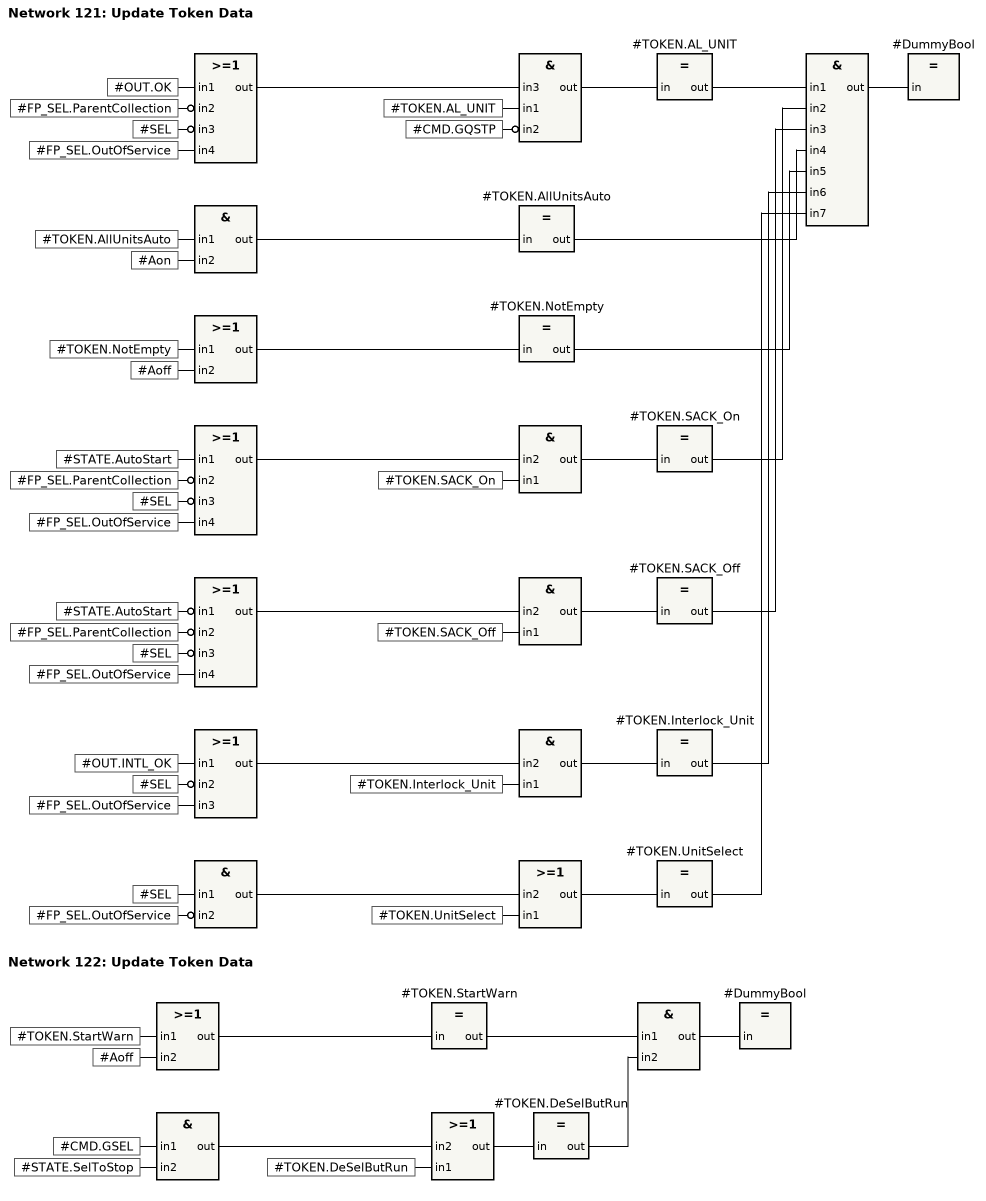
   #TOKEN.AL_UNIT := (#OUT.OK OR NOT #FP_SEL.ParentCollection OR NOT #SEL OR #FP_SEL.OutOfService) AND #TOKEN.AL_UNIT AND NOT #CMD.GQSTP;
   #TOKEN.SACK_On := (#STATE.AutoStart OR NOT #FP_SEL.ParentCollection OR NOT #SEL OR #FP_SEL.OutOfService) AND #TOKEN.SACK_On;
   #TOKEN.SACK_Off := (NOT #STATE.AutoStart OR NOT #FP_SEL.ParentCollection OR NOT #SEL OR #FP_SEL.OutOfService) AND #TOKEN.SACK_Off;
   #TOKEN.AllUnitsAuto := #TOKEN.AllUnitsAuto AND #Aon;
   #TOKEN.NotEmpty := #TOKEN.NotEmpty OR #Aoff;
   #TOKEN.Interlock_Unit := (#OUT.INTL_OK OR NOT #SEL OR #FP_SEL.OutOfService) AND #TOKEN.Interlock_Unit;
   #TOKEN.UnitSelect := (#SEL AND NOT #FP_SEL.OutOfService) OR #TOKEN.UnitSelect;
   #DummyBool := #TOKEN.AL_UNIT AND #TOKEN.SACK_On AND #TOKEN.SACK_Off AND #TOKEN.AllUnitsAuto AND #TOKEN.NotEmpty AND #TOKEN.Interlock_Unit AND #TOKEN.UnitSelect;
END_REGION

REGION Network 122: Update Token Data
   #TOKEN.StartWarn := #TOKEN.StartWarn OR #Aoff;
   #TOKEN.DeSelButRun := (#CMD.GSEL AND #STATE.SelToStop) OR #TOKEN.DeSelButRun;
   #DummyBool := #TOKEN.StartWarn AND #TOKEN.DeSelButRun;
END_REGION

REGION Network 123: Interlock Status to HMI
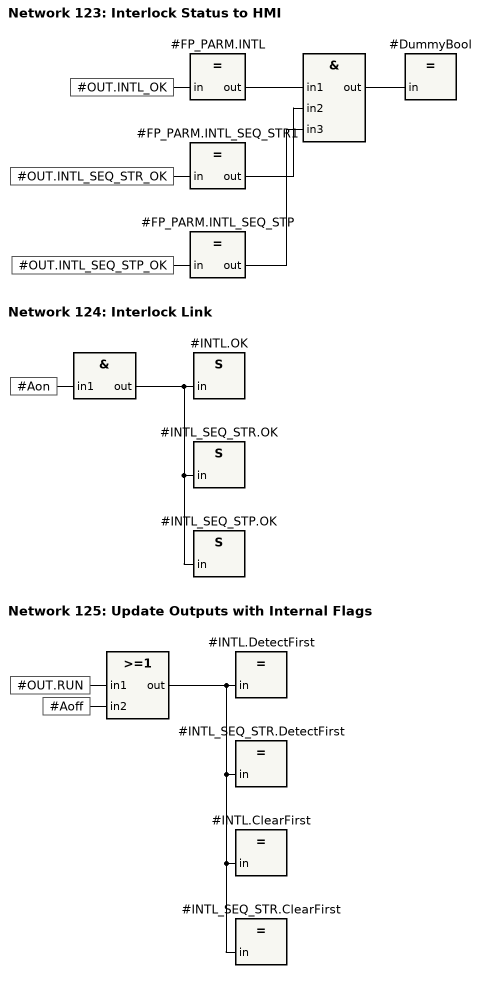
   #FP_PARM.INTL := #OUT.INTL_OK;
   #FP_PARM.INTL_SEQ_STR1 := #OUT.INTL_SEQ_STR_OK;
   #FP_PARM.INTL_SEQ_STP := #OUT.INTL_SEQ_STP_OK;
   #DummyBool := #OUT.INTL_OK AND #OUT.INTL_SEQ_STR_OK AND #OUT.INTL_SEQ_STP_OK;
END_REGION

REGION Network 124: Interlock Link
   IF #Aon THEN
       #INTL.OK := TRUE;
       #INTL_SEQ_STR.OK := TRUE;
       #INTL_SEQ_STP.OK := TRUE;
   END_IF;
END_REGION

REGION Network 125: Update Outputs with Internal Flags
   #INTL.DetectFirst := #OUT.RUN OR #Aoff;
   #INTL_SEQ_STR.DetectFirst := #INTL.DetectFirst;
   #INTL.ClearFirst := #INTL.DetectFirst;
   #INTL_SEQ_STR.ClearFirst := #INTL.DetectFirst;
END_REGION
END_FUNCTION_BLOCK

FUNCTION_BLOCK "ACESYS_BQ16_PROG"   // FB240, FBD
TITLE = ACESYS V8.0 - Build 002 - Air Blaster Program Block
{ S7_Optimized_Access := 'FALSE' }
AUTHOR : FLSmidth
FAMILY : ACESYS
NAME : Air_Prog
VERSION : 8.0
// This block is a separate program block for a airblaster and shall work as a 
// "child" for Air-blaster control block, ACESYS_BQ16_CTRL
// Data to the control block shall be send in a data structure: BQ16_Link (UDT224)
   VAR_OUTPUT
      Run : Bool;   // Program Running
      MSW : "ACESYS_HMI_STAT_32T";
   END_VAR
   VAR_IN_OUT
      TOKEN : "ACESYS_TOKEN";
      ProgLink : "ACESYS_BQ16";   // Link Command unit <-> Program Unit
   END_VAR
   VAR
      BlockInfo : Struct
         ACESYS_Version : Int;   // Block Version
         ACESYS_Build : Int;   // Block Build Number
         DB_Number : Int;
      END_STRUCT;
      FP_CMD : Struct   // Faceplate Commands
         Previous : Bool;   // FacePlateCmd (bit 8): Previous Sequence
         Next : Bool;   // FacePlateCmd (bit 9): Next Sequence
         Spare_Bool_01 : Bool;   // FacePlateCmd (bit 10): Spare
         Spare_Bool_02 : Bool;   // FacePlateCmd (bit 11): Spare
         Spare_Bool_03 : Bool;   // FacePlateCmd (bit 12): Spare
         Spare_Bool_04 : Bool;   // FacePlateCmd (bit 13): Spare
         Spare_Bool_05 : Bool;   // FacePlateCmd (bit 14): Spare
         Spare_Bool_06 : Bool;   // FacePlateCmd (bit 15): ECS Acknowledge
         Spare_Bool_07 : Bool;   // FacePlateCmd (bit 0): Spare
         Spare_Bool_08 : Bool;   // FacePlateCmd (bit 1): Spare
         Spare_Bool_09 : Bool;   // FacePlateCmd (bit 2): Spare
         Spare_Bool_10 : Bool;   // FacePlateCmd (bit 3): Spare
         Spare_Bool_11 : Bool;   // FacePlateCmd (bit 4): Spare
         Spare_Bool_12 : Bool;   // FacePlateCmd (bit 5): Spare
         Spare_Bool_13 : Bool;   // FacePlateCmd (bit 6): Spare
         Spare_Bool_14 : Bool;   // FacePlateCmd (bit 7): Spare
      END_STRUCT;
      FP_DIM : Struct   // Faceplate Dimmed Buttons
         Previous : Bool;   // Dimout Prev button to ECS
         Next : Bool;   // Dimout Next button to ECS
         Spare_Bool_01 : Bool;
         Spare_Bool_02 : Bool;
         Spare_Bool_03 : Bool;
         Spare_Bool_04 : Bool;
         Spare_Bool_05 : Bool;
         Spare_Bool_06 : Bool;
         Spare_Bool_07 : Bool;
         Spare_Bool_08 : Bool;
         Spare_Bool_09 : Bool;
         Spare_Bool_10 : Bool;
         Spare_Bool_11 : Bool;
         Spare_Bool_12 : Bool;
         Spare_Bool_13 : Bool;
         Spare_Bool_14 : Bool;
      END_STRUCT;
      FP_PARM : Struct
         ProgNo : Int;   // Program Number to Faceplate
         SEQNO : Int;   // Sequence No in Matrix Configuration Faceplate
         NumberBlasters : Int := 16;   // Number Of Blasters to be Used
         NumberSteps : Int := 16;   // Number Of Steps to be Used
         Blast_Stp_Dyn01 : Bool;   // Blaster 1 Setup Dynamic bit to ECS
         Blast_Stp_Dyn02 : Bool;   // Blaster 2 Setup Dynamic bit to ECS
         Blast_Stp_Dyn03 : Bool;   // Blaster 3 Setup Dynamic bit to ECS
         Blast_Stp_Dyn04 : Bool;   // Blaster 4 Setup Dynamic bit to ECS
         Blast_Stp_Dyn05 : Bool;   // Blaster 5 Setup Dynamic bit to ECS
         Blast_Stp_Dyn06 : Bool;   // Blaster 6 Setup Dynamic bit to ECS
         Blast_Stp_Dyn07 : Bool;   // Blaster 7 Setup Dynamic bit to ECS
         Blast_Stp_Dyn08 : Bool;   // Blaster 8 Setup Dynamic bit to ECS
         Blast_Stp_Dyn09 : Bool;   // Blaster 9 Setup Dynamic bit to ECS
         Blast_Stp_Dyn10 : Bool;   // Blaster 10 Setup Dynamic bit to ECS
         Blast_Stp_Dyn11 : Bool;   // Blaster 11 Setup Dynamic bit to ECS
         Blast_Stp_Dyn12 : Bool;   // Blaster 12 Setup Dynamic bit to ECS
         Blast_Stp_Dyn13 : Bool;   // Blaster 13 Setup Dynamic bit to ECS
         Blast_Stp_Dyn14 : Bool;   // Blaster 14 Setup Dynamic bit to ECS
         Blast_Stp_Dyn15 : Bool;   // Blaster 15 Setup Dynamic bit to ECS
         Blast_Stp_Dyn16 : Bool;   // Blaster 16 Setup Dynamic bit to ECS
         CurrentState : Array[1..16] of Int;   // Blaster State for ECS animation
      END_STRUCT;
      FP_PARM_CycleTime : Array[1..6] of Int;   // SP from FP
      FP_PARM_OffsetTime : Array[1..6] of Int;   // SP from FP
      FP_PARM_PulseTime : Array[1..6] of Int;   // SP from FP
      FP_PARM_StepTime : Array[1..6] of Int;   // SP from FP
      FP_PARM_Blaster_SEQNO : Array[1..16] of Int;   // Blaster Configured Sequence
      FP_PARM_BlastSEQX_Setup : Array[1..16] of Word;   // Blaster Setup From/To ECS
      FP_PARM_Blaster_Step : Array[1..16] of Word;   // Blaster Configurated Step Mask
      FP_PARM_MaxNumberSteps : Array[1..16] of Int;   // Max Step to be executed with current Time constants
      FP_PARM_PauseTime : Array[1..16] of Int;   // Time until next Cycle
      FP_PARM_MaxStep : Array[1..6] of Int;   // Max Step to be executed with current Time constants
      FP_PARM_OffsetStep : Array[1..16] of Bool;
      BlastSEQ1_Setup : Array[1..16] of Word;   // Blaster Setup in sequence 01
      BlastSEQ2_Setup : Array[1..16] of Word;   // Blaster Setup in sequence 02
      BlastSEQ3_Setup : Array[1..16] of Word;   // Blaster Setup in sequence 03
      BlastSEQ4_Setup : Array[1..16] of Word;   // Blaster Setup in sequence 04
      BlastSEQ5_Setup : Array[1..16] of Word;   // Blaster Setup in sequence 05
      BlastSEQ6_Setup : Array[1..16] of Word;   // Blaster Setup in sequence 06
      BlastSEQ_CycleTime_Mem : Array[1..6] of Int;   // Internal Timer Value
      BlastSEQ_CycleTime_PV : Array[1..6] of Int;   // For Next Blast, Time Calculation
      StepTime_PV : Array[1..6] of Int;   // For Next Blast, Time Calculation
      SEQTmr_SP : Array[1..6] of Int;   // For Next Blast, Time Calculation
      BlastSEQ_State : Array[1..6] of Word;   // Actual Step Mask of the Sequence
      TimeACT_PV : Array[1..6] of Int;   // For Next Blast, Time Calculation
      PauseTime : Array[1..6] of Int;   // Time until next Cycle
      BlastSEQ_CycleTime_DN : Array[1..6] of Bool;   // Timer Done
      StepSEQ_Offset : Array[1..6] of Bool;   // Select Offset time
      StepSEQ_Pulse : Array[1..6] of Bool;   // Select Pulse Time
      StepSEQ_Step : Array[1..6] of Bool;   // Select Step Time
      StepSEQ_Done : Array[1..6] of Bool;   // Step Sequence Done
      BlastSEQ_Start : Array[1..6] of Bool;   // Start Sequence
      BlastSEQ_EN : Array[1..6] of Bool;   // Pause the Execution of sequence
      InOffset_Pause : Array[1..6] of Bool;   // Pause the Execution of sequence
      CycleInStep : Array[1..6] of Bool;   // Cycle is running a step
      SequenceInOffset : Array[1..6] of Bool;   // Sequence is in Offset state
      TimeOLD : Array[1..6] of Time;
      TimeACT : Array[1..6] of Time;
      TimeSP : Array[1..6] of Time;
      SEQ_Old_Config : Array[1..6] of DWord;
      CycleTime_Old : Array[1..6] of Int;
      OffsetTime_Old : Array[1..6] of Int;
      PulseTime_Old : Array[1..6] of Int;
      StepTime_Old : Array[1..6] of Int;
      ConfigChanged : Bool;   // Configuration Changed Status
      ProgLink_Start : Bool;   // Start from Control Block
      ProgLink_Reset : Bool;   // Reset Sequence Option from Control Block
      Run_Delay : Bool;   // One scan delayed RUN signal
      SEQ01_Timer_DN : Bool;
      SEQ02_Timer_DN : Bool;
      SEQ03_Timer_DN : Bool;
      SEQ04_Timer_DN : Bool;
      SEQ05_Timer_DN : Bool;
      SEQ06_Timer_DN : Bool;
      Old_SEQNO : Int;
      StatusWork : Int;
      MSW_Status : Int;
      SYNC_TIME : Struct
         Mem : Int;
         PRE : Int;
         PRE_Old : Int;
         PV : Int;
         DN : Bool;
         TT : Bool;
      END_STRUCT;
      CMD_Int : Struct
         Previous : Bool;
         Next : Bool;
      END_STRUCT;
      ONS : Struct
         Previous : Bool;
         Next : Bool;
         Pulse : Array[1..6] of Bool;   // Pause the Execution of sequence
         Pulse1 : Array[1..6] of Bool;   // Pause the Execution of sequence
         ConfigChanged : Bool;
         BlastSEQ01_Start : Bool;
         BlastSEQ02_Start : Bool;
         BlastSEQ03_Start : Bool;
         BlastSEQ04_Start : Bool;
         BlastSEQ05_Start : Bool;
         BlastSEQ06_Start : Bool;
         Sync_Time_DN : Bool;
      END_STRUCT;
      OUT : Struct
         Run : Bool;
      END_STRUCT;
      SEQ01_Timer : TON_TIME;
      SEQ02_Timer : TON_TIME;
      SEQ03_Timer : TON_TIME;
      SEQ04_Timer : TON_TIME;
      SEQ05_Timer : TON_TIME;
      SEQ06_Timer : TON_TIME;
   END_VAR
   VAR_TEMP
      Aon : Bool;
      Aoff : Bool;
      DummyBool : Bool;
      DummyBool1 : Bool;
      DummyTime : Time;
      DummyWord : Word;
      DummyDint : DInt;
      DummyInt : Int;
      DummyReal : Real;
      DummyReal1 : Real;
      Current_SEQNO : Int;
      NextTime_BlastLoop : Int;
      Offset_Int : Int;
      NXT_SEQ_State : Word;   // Current Step Mask of the Sequence
      NXT_SEQ_PULSE : Bool;
      SEQ_Current_Config : Array[1..6] of DWord;
      ClearBlasterLoop : Int;
      ClearStepLoop : Int;
      StepMask : Word;   // Allowed Steps set to 1
      ChangeConfigLoop : Int;
   END_VAR
   VAR_TEMP   // added for the SCL form of the ladder/FBD networks
      _w1 : Bool;
      _w2 : Bool;
      _w3 : Bool;
      _w4 : Bool;
      _w5 : Bool;
      _w6 : Bool;
      _w7 : Bool;
      _w8 : Bool;
      _w9 : Bool;
      _w10 : Bool;
      _w11 : Bool;
      _w12 : Bool;
      _w13 : Bool;
      _w14 : Bool;
      _w15 : Bool;
      _w16 : Bool;
   END_VAR
   // FP_PARM_CycleTime[1] := 1;
   // FP_PARM_CycleTime[2] := 1;
   // FP_PARM_CycleTime[3] := 1;
   // FP_PARM_CycleTime[4] := 1;
   // FP_PARM_CycleTime[5] := 1;
   // FP_PARM_CycleTime[6] := 1;
   // FP_PARM_OffsetTime[1] := 30;
   // FP_PARM_OffsetTime[2] := 30;
   // FP_PARM_OffsetTime[3] := 30;
   // FP_PARM_OffsetTime[4] := 30;
   // FP_PARM_OffsetTime[5] := 30;
   // FP_PARM_OffsetTime[6] := 30;
   // FP_PARM_PulseTime[1] := 500;
   // FP_PARM_PulseTime[2] := 500;
   // FP_PARM_PulseTime[3] := 500;
   // FP_PARM_PulseTime[4] := 500;
   // FP_PARM_PulseTime[5] := 500;
   // FP_PARM_PulseTime[6] := 500;
   // FP_PARM_StepTime[1] := 5;
   // FP_PARM_StepTime[2] := 5;
   // FP_PARM_StepTime[3] := 5;
   // FP_PARM_StepTime[4] := 5;
   // FP_PARM_StepTime[5] := 5;
   // FP_PARM_StepTime[6] := 5;
BEGIN

REGION Network 1: Aon/Aoff Definition
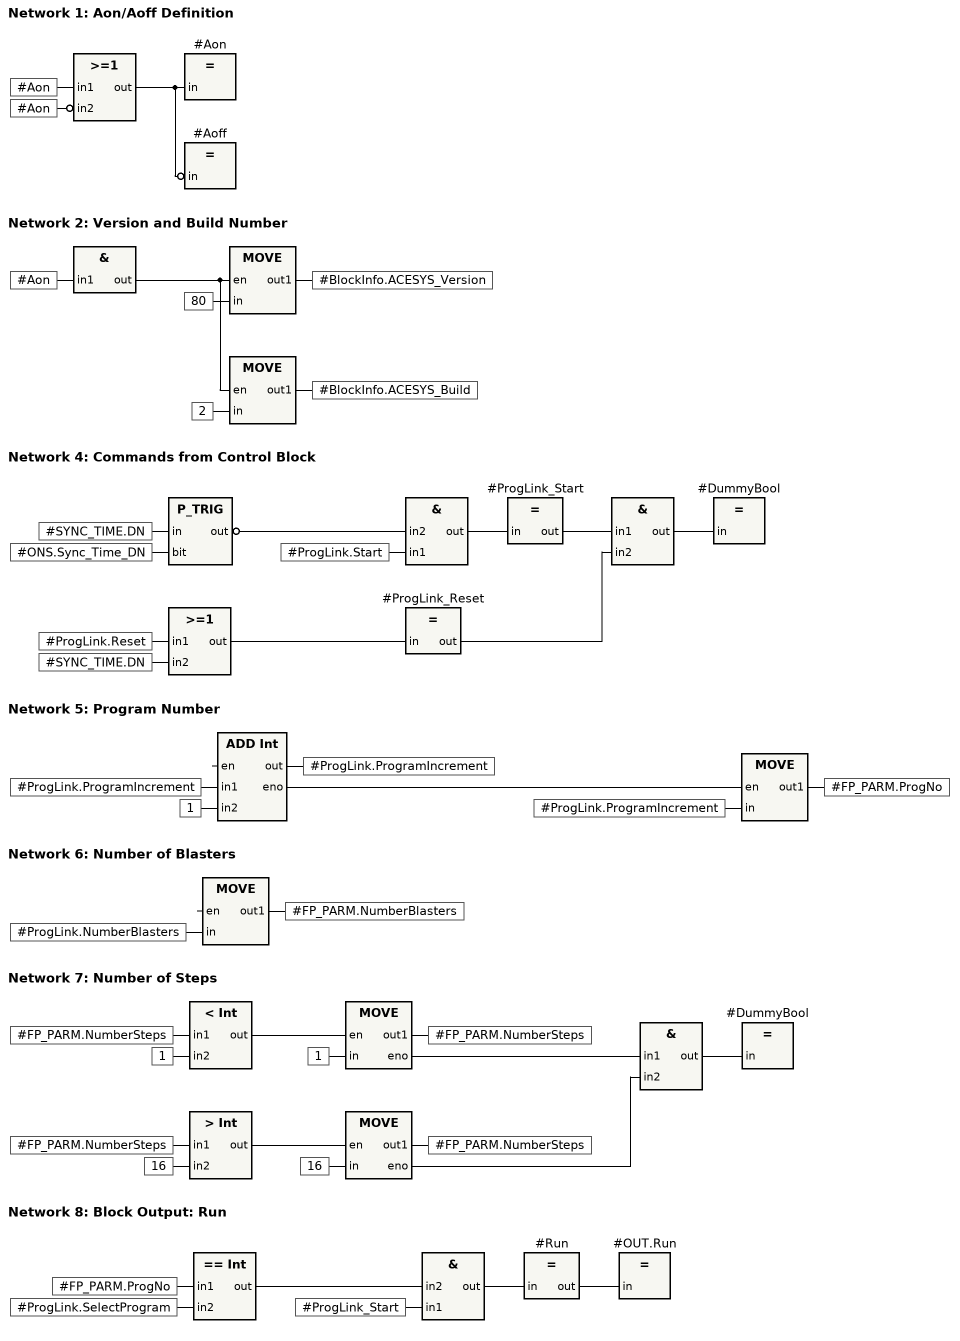
   #Aon := #Aon OR NOT #Aon;
   #Aoff := NOT #Aon;
END_REGION

REGION Network 2: Version and Build Number
   IF #Aon THEN
       #BlockInfo.ACESYS_Version := 80;
       #BlockInfo.ACESYS_Build := 2;
   END_IF;
END_REGION

REGION Network 3 (STL): Instance DB Number to Faceplate
         L     DINO;
         T     #BlockInfo.DB_Number;
END_REGION

REGION Network 4: Commands from Control Block
   // Introduce Sync Timer to reinitialize all sequences
   #_w1 := #SYNC_TIME.DN AND NOT #ONS.Sync_Time_DN;   // rising edge
   #ONS.Sync_Time_DN := #SYNC_TIME.DN;
   #ProgLink_Start := NOT #_w1 AND #ProgLink.Start;
   #ProgLink_Reset := #ProgLink.Reset OR #SYNC_TIME.DN;
   #DummyBool := #ProgLink_Start AND #ProgLink_Reset;
END_REGION

REGION Network 5: Program Number
   // Increment program counter in each instance block
   // ENO of a box is taken as its EN; it also drops when the box reports an error
   #ProgLink.ProgramIncrement := #ProgLink.ProgramIncrement + 1;
   #FP_PARM.ProgNo := #ProgLink.ProgramIncrement;
END_REGION

REGION Network 6: Number of Blasters
   #FP_PARM.NumberBlasters := #ProgLink.NumberBlasters;
END_REGION

REGION Network 7: Number of Steps
   // Allowed range 1 - 16
   // ENO of a box is taken as its EN; it also drops when the box reports an error
   #_w1 := #FP_PARM.NumberSteps < 1;
   IF #_w1 THEN #FP_PARM.NumberSteps := 1; END_IF;
   #_w2 := #FP_PARM.NumberSteps > 16;
   IF #_w2 THEN #FP_PARM.NumberSteps := 16; END_IF;
   #DummyBool := #_w1 AND #_w2;
END_REGION

REGION Network 8: Block Output: Run
   #Run := (#FP_PARM.ProgNo = #ProgLink.SelectProgram) AND #ProgLink_Start;
   #OUT.Run := #Run;
END_REGION

REGION Network 9: Dimout Faceplate Pushbuttons
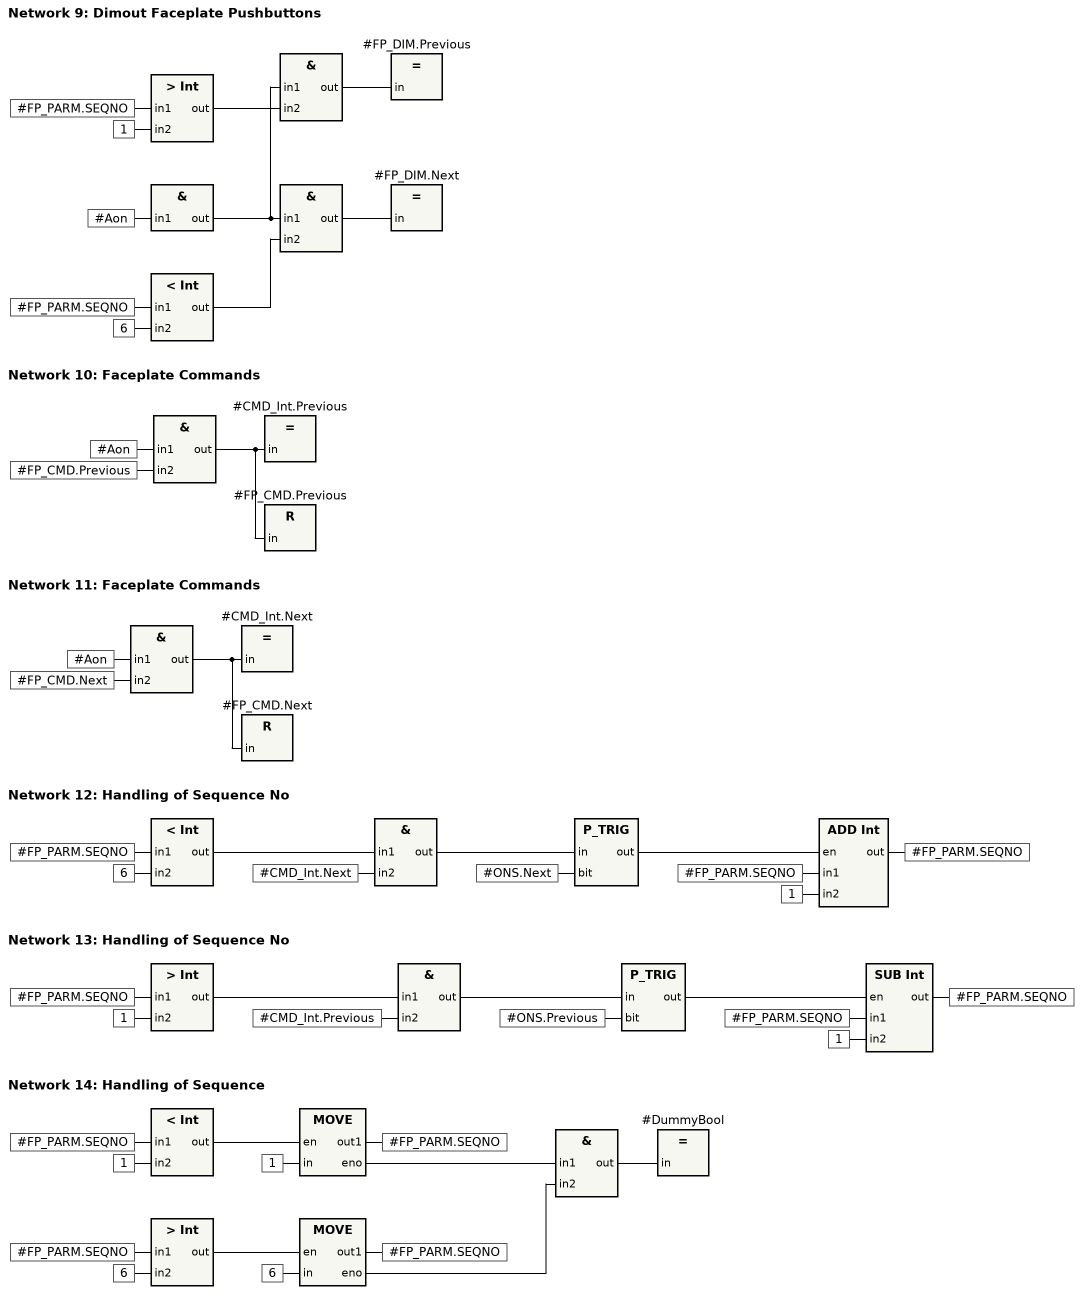
   #FP_DIM.Previous := #Aon AND (#FP_PARM.SEQNO > 1);
   #FP_DIM.Next := #Aon AND (#FP_PARM.SEQNO < 6);
END_REGION

REGION Network 10: Faceplate Commands
   #CMD_Int.Previous := #Aon AND #FP_CMD.Previous;
   IF #CMD_Int.Previous THEN #FP_CMD.Previous := FALSE; END_IF;
END_REGION

REGION Network 11: Faceplate Commands
   #CMD_Int.Next := #Aon AND #FP_CMD.Next;
   IF #CMD_Int.Next THEN #FP_CMD.Next := FALSE; END_IF;
END_REGION

REGION Network 12: Handling of Sequence No
   // Incrementing the SEQ NO
   #_w1 := (#FP_PARM.SEQNO < 6) AND #CMD_Int.Next;
   #_w2 := #_w1 AND NOT #ONS.Next;   // rising edge
   #ONS.Next := #_w1;
   IF #_w2 THEN #FP_PARM.SEQNO := #FP_PARM.SEQNO + 1; END_IF;
END_REGION

REGION Network 13: Handling of Sequence No
   // Decrementing the SEQ NO
   #_w1 := (#FP_PARM.SEQNO > 1) AND #CMD_Int.Previous;
   #_w2 := #_w1 AND NOT #ONS.Previous;   // rising edge
   #ONS.Previous := #_w1;
   IF #_w2 THEN #FP_PARM.SEQNO := #FP_PARM.SEQNO - 1; END_IF;
END_REGION

REGION Network 14: Handling of Sequence
   // Keep sequence number in range
   // ENO of a box is taken as its EN; it also drops when the box reports an error
   #_w1 := #FP_PARM.SEQNO < 1;
   IF #_w1 THEN #FP_PARM.SEQNO := 1; END_IF;
   #_w2 := #FP_PARM.SEQNO > 6;
   IF #_w2 THEN #FP_PARM.SEQNO := 6; END_IF;
   #DummyBool := #_w1 AND #_w2;
END_REGION

REGION Network 15: Maximum Step in Sequence #1 to be Executed with Current Time Constants
   // (CycleTime) / (PulseTime + StepTime)
   // Truncate result to get #of FULL steps contained in configured Cycle Time
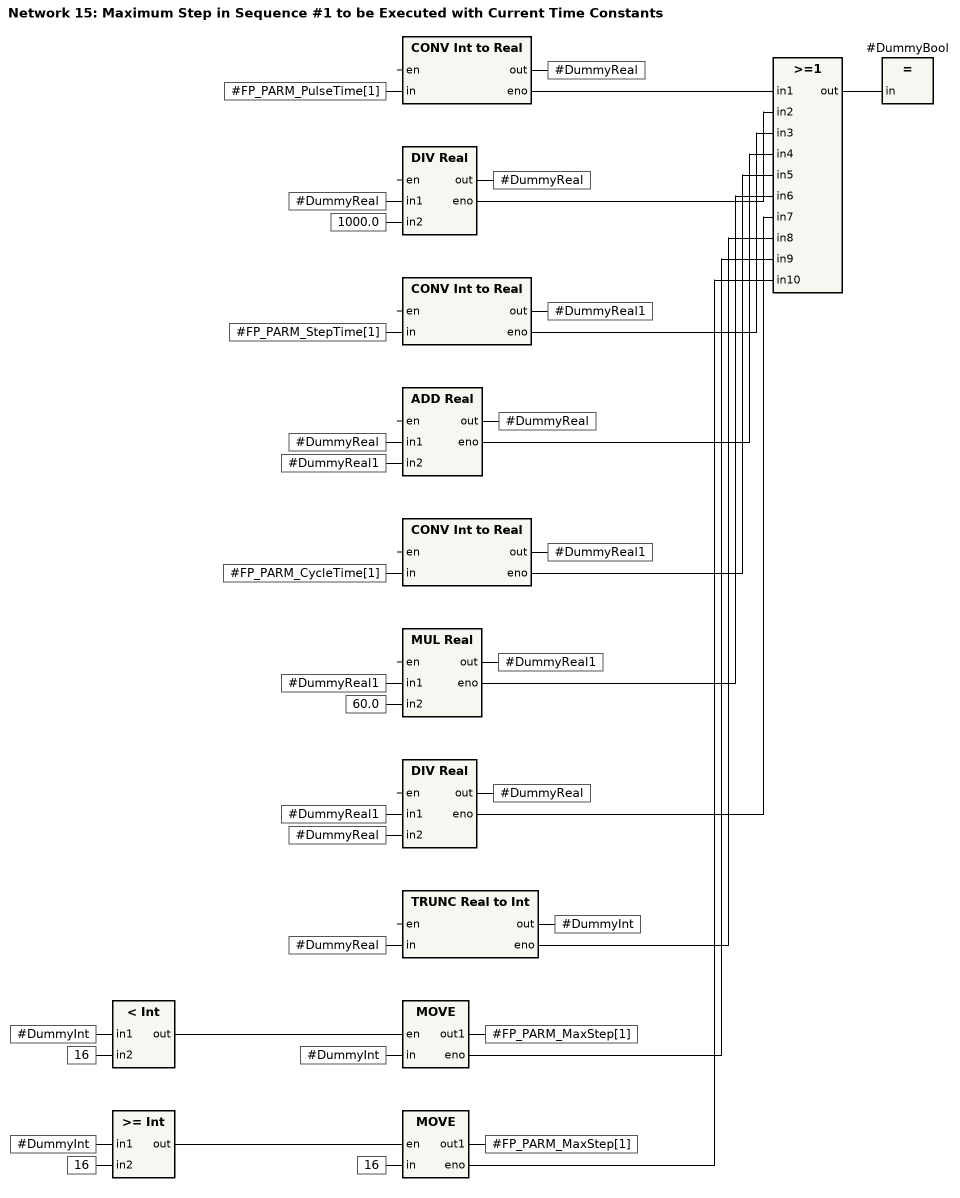
   #DummyReal := INT_TO_REAL(#FP_PARM_PulseTime[1]);
   #DummyReal := #DummyReal / 1000.0;
   #DummyReal1 := INT_TO_REAL(#FP_PARM_StepTime[1]);
   #DummyReal := #DummyReal + #DummyReal1;
   #DummyReal1 := INT_TO_REAL(#FP_PARM_CycleTime[1]);
   #DummyReal1 := #DummyReal1 * 60.0;
   #DummyReal := #DummyReal1 / #DummyReal;
   #DummyInt := TRUNC(#DummyReal);
   #_w1 := #DummyInt < 16;
   IF #_w1 THEN #FP_PARM_MaxStep[1] := #DummyInt; END_IF;
   #_w2 := #DummyInt >= 16;
   IF #_w2 THEN #FP_PARM_MaxStep[1] := 16; END_IF;
   #DummyBool := TRUE OR TRUE OR TRUE OR TRUE OR TRUE OR TRUE OR TRUE OR TRUE OR #_w1 OR #_w2;
END_REGION

REGION Network 16: Maximum Step in Sequence #2 to be Executed with Current Time Constants
   // (CycleTime) / (PulseTime + StepTime)
   // Truncate result to get #of FULL steps contained in configured Cycle Time
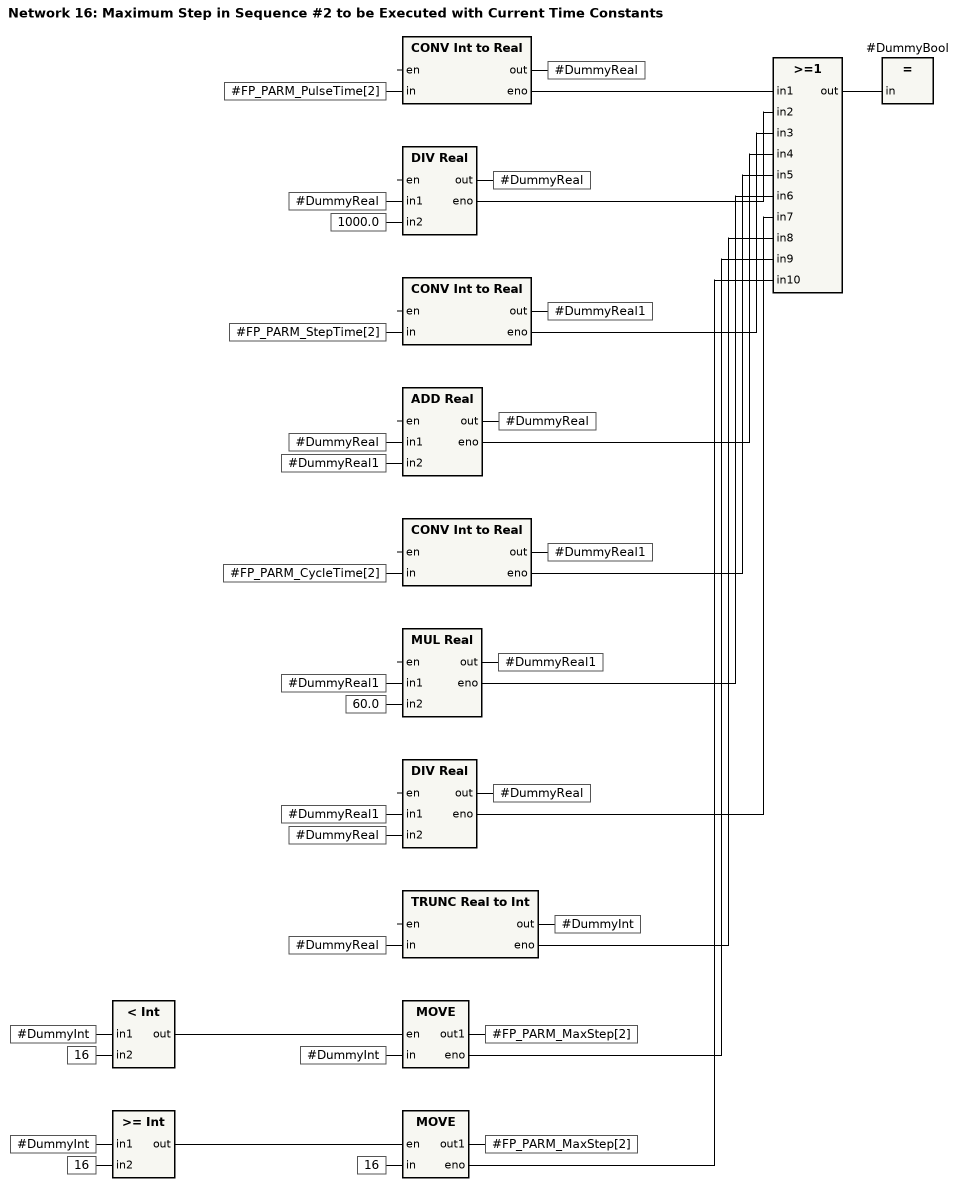
   #DummyReal := INT_TO_REAL(#FP_PARM_PulseTime[2]);
   #DummyReal := #DummyReal / 1000.0;
   #DummyReal1 := INT_TO_REAL(#FP_PARM_StepTime[2]);
   #DummyReal := #DummyReal + #DummyReal1;
   #DummyReal1 := INT_TO_REAL(#FP_PARM_CycleTime[2]);
   #DummyReal1 := #DummyReal1 * 60.0;
   #DummyReal := #DummyReal1 / #DummyReal;
   #DummyInt := TRUNC(#DummyReal);
   #_w1 := #DummyInt < 16;
   IF #_w1 THEN #FP_PARM_MaxStep[2] := #DummyInt; END_IF;
   #_w2 := #DummyInt >= 16;
   IF #_w2 THEN #FP_PARM_MaxStep[2] := 16; END_IF;
   #DummyBool := TRUE OR TRUE OR TRUE OR TRUE OR TRUE OR TRUE OR TRUE OR TRUE OR #_w1 OR #_w2;
END_REGION

REGION Network 17: Maximum Step in Sequence #3 to be Executed with Current Time Constants
   // (CycleTime) / (PulseTime + StepTime)
   // Truncate result to get #of FULL steps contained in configured Cycle Time
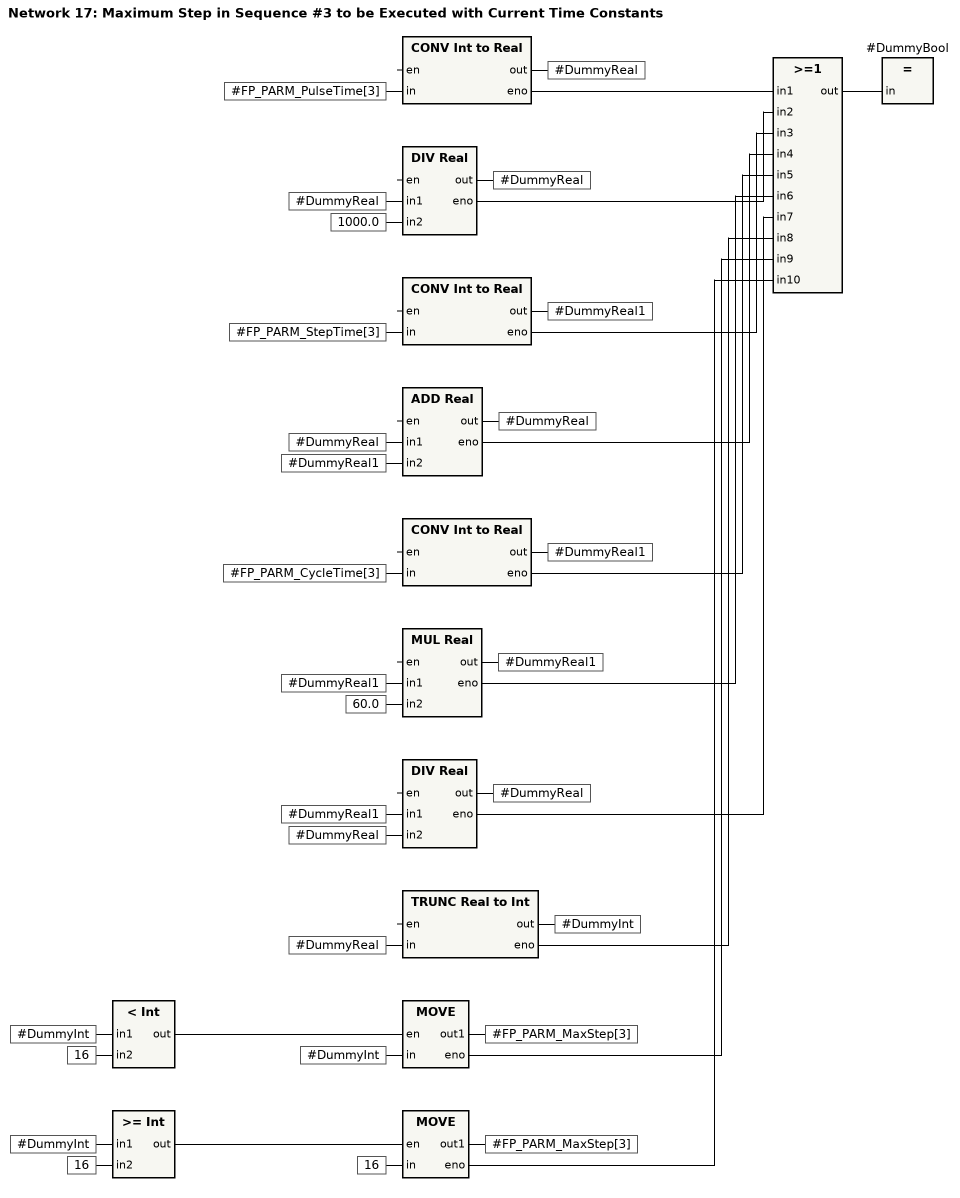
   #DummyReal := INT_TO_REAL(#FP_PARM_PulseTime[3]);
   #DummyReal := #DummyReal / 1000.0;
   #DummyReal1 := INT_TO_REAL(#FP_PARM_StepTime[3]);
   #DummyReal := #DummyReal + #DummyReal1;
   #DummyReal1 := INT_TO_REAL(#FP_PARM_CycleTime[3]);
   #DummyReal1 := #DummyReal1 * 60.0;
   #DummyReal := #DummyReal1 / #DummyReal;
   #DummyInt := TRUNC(#DummyReal);
   #_w1 := #DummyInt < 16;
   IF #_w1 THEN #FP_PARM_MaxStep[3] := #DummyInt; END_IF;
   #_w2 := #DummyInt >= 16;
   IF #_w2 THEN #FP_PARM_MaxStep[3] := 16; END_IF;
   #DummyBool := TRUE OR TRUE OR TRUE OR TRUE OR TRUE OR TRUE OR TRUE OR TRUE OR #_w1 OR #_w2;
END_REGION

REGION Network 18: Maximum Step in Sequence #4 to be Executed with Current Time Constants
   // (CycleTime) / (PulseTime + StepTime)
   // Truncate result to get #of FULL steps contained in configured Cycle Time
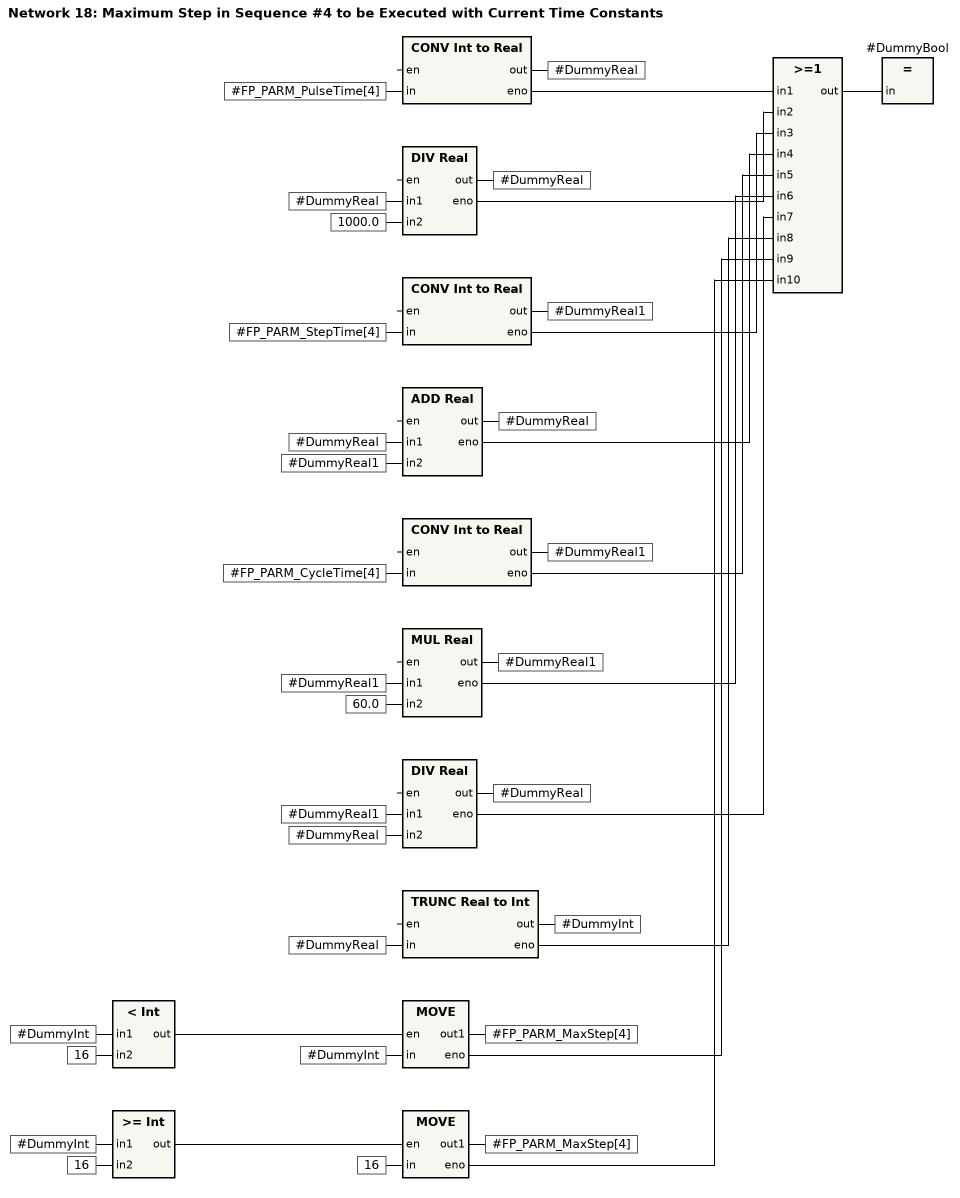
   #DummyReal := INT_TO_REAL(#FP_PARM_PulseTime[4]);
   #DummyReal := #DummyReal / 1000.0;
   #DummyReal1 := INT_TO_REAL(#FP_PARM_StepTime[4]);
   #DummyReal := #DummyReal + #DummyReal1;
   #DummyReal1 := INT_TO_REAL(#FP_PARM_CycleTime[4]);
   #DummyReal1 := #DummyReal1 * 60.0;
   #DummyReal := #DummyReal1 / #DummyReal;
   #DummyInt := TRUNC(#DummyReal);
   #_w1 := #DummyInt < 16;
   IF #_w1 THEN #FP_PARM_MaxStep[4] := #DummyInt; END_IF;
   #_w2 := #DummyInt >= 16;
   IF #_w2 THEN #FP_PARM_MaxStep[4] := 16; END_IF;
   #DummyBool := TRUE OR TRUE OR TRUE OR TRUE OR TRUE OR TRUE OR TRUE OR TRUE OR #_w1 OR #_w2;
END_REGION

REGION Network 19: Maximum Step in Sequence #5 to be Executed with Current Time Constants
   // (CycleTime) / (PulseTime + StepTime)
   // Truncate result to get #of FULL steps contained in configured Cycle Time
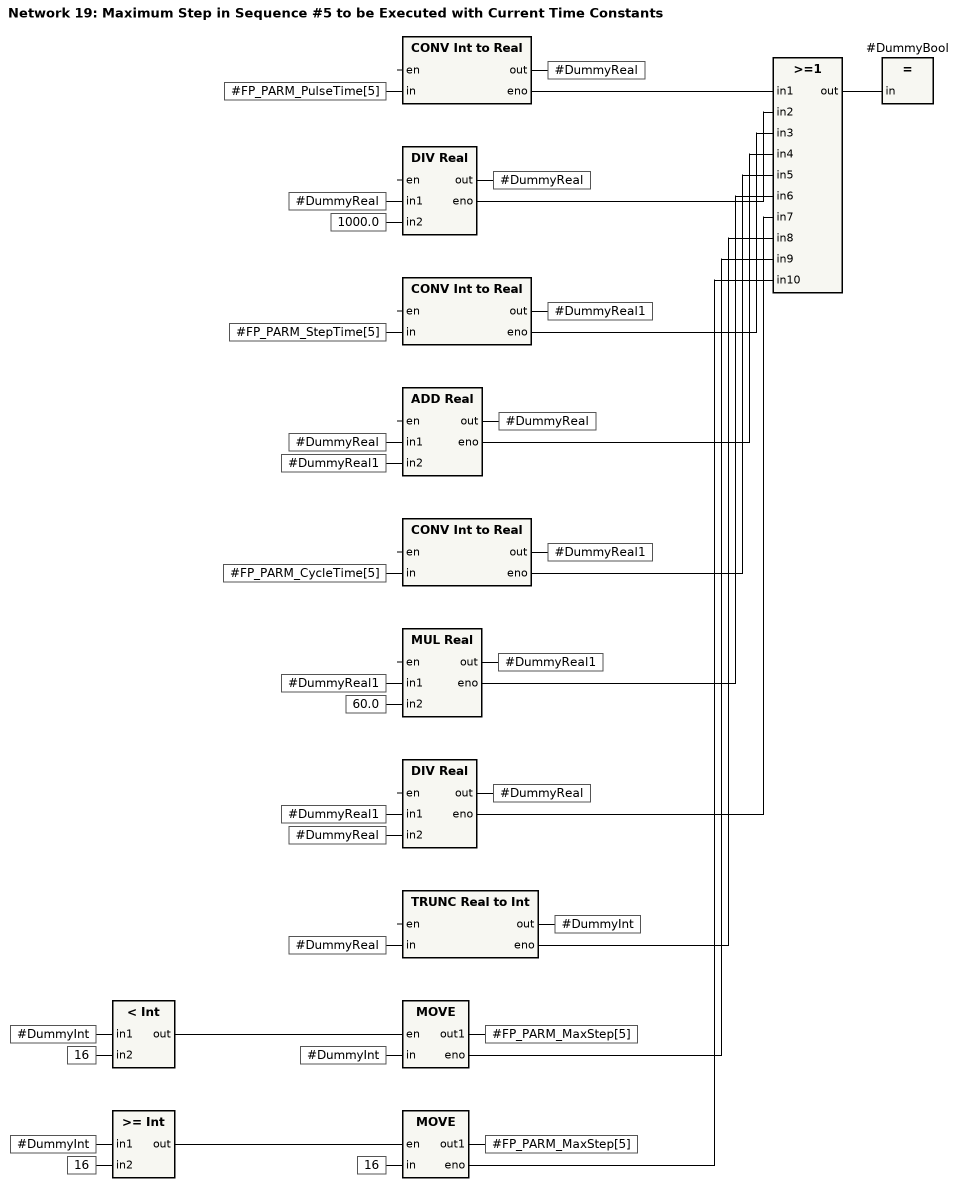
   #DummyReal := INT_TO_REAL(#FP_PARM_PulseTime[5]);
   #DummyReal := #DummyReal / 1000.0;
   #DummyReal1 := INT_TO_REAL(#FP_PARM_StepTime[5]);
   #DummyReal := #DummyReal + #DummyReal1;
   #DummyReal1 := INT_TO_REAL(#FP_PARM_CycleTime[5]);
   #DummyReal1 := #DummyReal1 * 60.0;
   #DummyReal := #DummyReal1 / #DummyReal;
   #DummyInt := TRUNC(#DummyReal);
   #_w1 := #DummyInt < 16;
   IF #_w1 THEN #FP_PARM_MaxStep[5] := #DummyInt; END_IF;
   #_w2 := #DummyInt >= 16;
   IF #_w2 THEN #FP_PARM_MaxStep[5] := 16; END_IF;
   #DummyBool := TRUE OR TRUE OR TRUE OR TRUE OR TRUE OR TRUE OR TRUE OR TRUE OR #_w1 OR #_w2;
END_REGION

REGION Network 20: Maximum Step in Sequence #6 to be Executed with Current Time Constants
   // (CycleTime) / (PulseTime + StepTime)
   // Truncate result to get #of FULL steps contained in configured Cycle Time
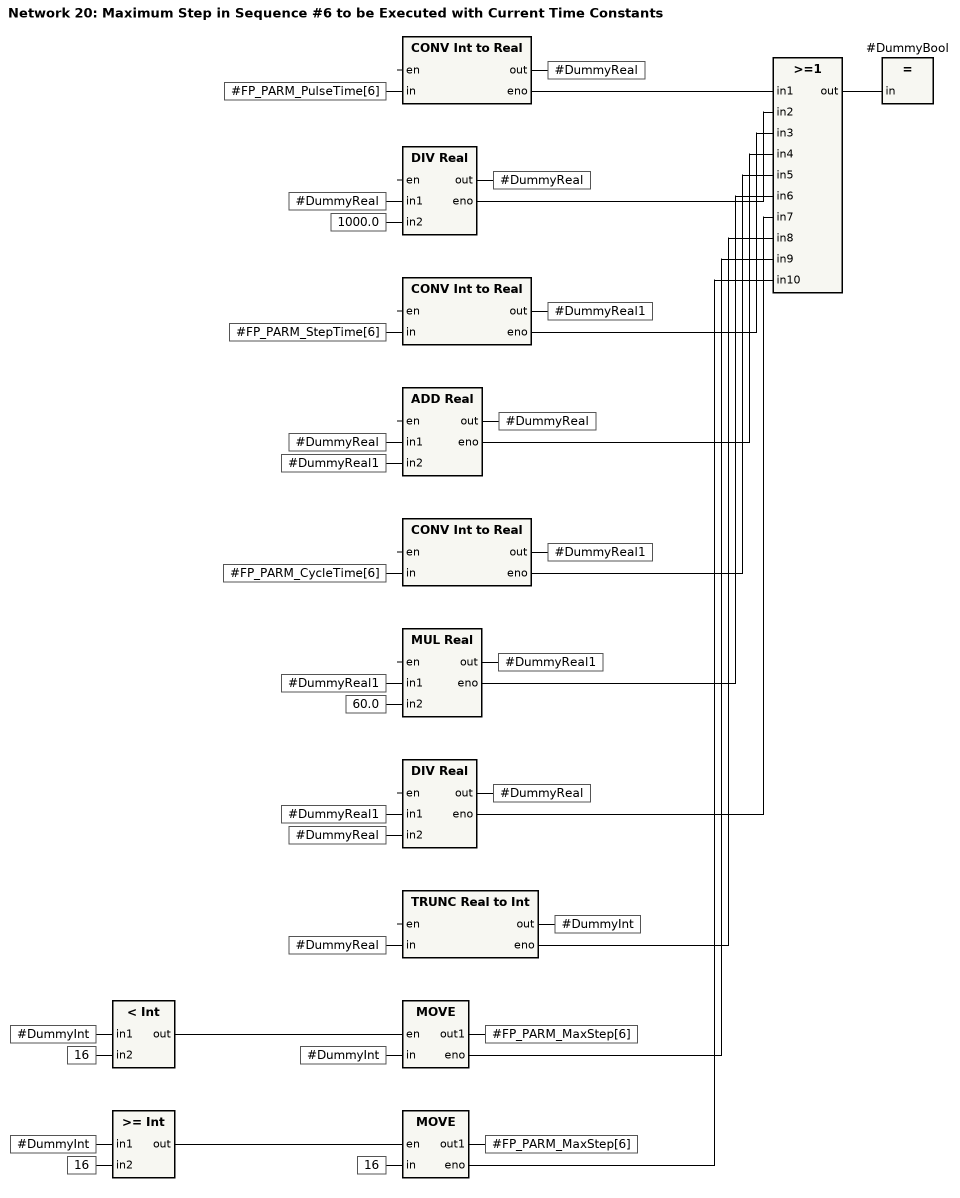
   #DummyReal := INT_TO_REAL(#FP_PARM_PulseTime[6]);
   #DummyReal := #DummyReal / 1000.0;
   #DummyReal1 := INT_TO_REAL(#FP_PARM_StepTime[6]);
   #DummyReal := #DummyReal + #DummyReal1;
   #DummyReal1 := INT_TO_REAL(#FP_PARM_CycleTime[6]);
   #DummyReal1 := #DummyReal1 * 60.0;
   #DummyReal := #DummyReal1 / #DummyReal;
   #DummyInt := TRUNC(#DummyReal);
   #_w1 := #DummyInt < 16;
   IF #_w1 THEN #FP_PARM_MaxStep[6] := #DummyInt; END_IF;
   #_w2 := #DummyInt >= 16;
   IF #_w2 THEN #FP_PARM_MaxStep[6] := 16; END_IF;
   #DummyBool := TRUE OR TRUE OR TRUE OR TRUE OR TRUE OR TRUE OR TRUE OR TRUE OR #_w1 OR #_w2;
END_REGION

REGION Network 21: Pause Time Sequence #1
   // Time between last step and cycle restart.
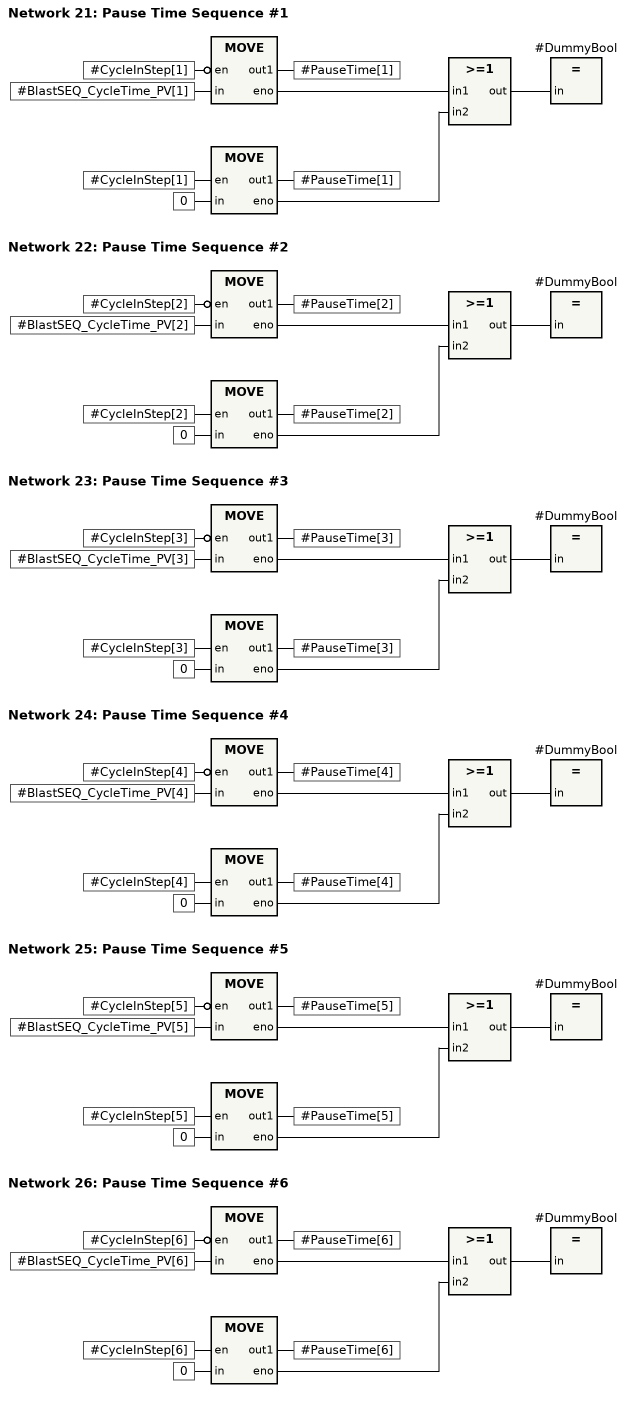
   IF NOT #CycleInStep[1] THEN #PauseTime[1] := #BlastSEQ_CycleTime_PV[1]; END_IF;
   IF #CycleInStep[1] THEN #PauseTime[1] := 0; END_IF;
   #DummyBool := NOT #CycleInStep[1] OR #CycleInStep[1];
END_REGION

REGION Network 22: Pause Time Sequence #2
   // Time between last step and cycle restart.
   IF NOT #CycleInStep[2] THEN #PauseTime[2] := #BlastSEQ_CycleTime_PV[2]; END_IF;
   IF #CycleInStep[2] THEN #PauseTime[2] := 0; END_IF;
   #DummyBool := NOT #CycleInStep[2] OR #CycleInStep[2];
END_REGION

REGION Network 23: Pause Time Sequence #3
   // Time between last step and cycle restart.
   IF NOT #CycleInStep[3] THEN #PauseTime[3] := #BlastSEQ_CycleTime_PV[3]; END_IF;
   IF #CycleInStep[3] THEN #PauseTime[3] := 0; END_IF;
   #DummyBool := NOT #CycleInStep[3] OR #CycleInStep[3];
END_REGION

REGION Network 24: Pause Time Sequence #4
   // Time between last step and cycle restart.
   IF NOT #CycleInStep[4] THEN #PauseTime[4] := #BlastSEQ_CycleTime_PV[4]; END_IF;
   IF #CycleInStep[4] THEN #PauseTime[4] := 0; END_IF;
   #DummyBool := NOT #CycleInStep[4] OR #CycleInStep[4];
END_REGION

REGION Network 25: Pause Time Sequence #5
   // Time between last step and cycle restart.
   IF NOT #CycleInStep[5] THEN #PauseTime[5] := #BlastSEQ_CycleTime_PV[5]; END_IF;
   IF #CycleInStep[5] THEN #PauseTime[5] := 0; END_IF;
   #DummyBool := NOT #CycleInStep[5] OR #CycleInStep[5];
END_REGION

REGION Network 26: Pause Time Sequence #6
   // Time between last step and cycle restart.
   IF NOT #CycleInStep[6] THEN #PauseTime[6] := #BlastSEQ_CycleTime_PV[6]; END_IF;
   IF #CycleInStep[6] THEN #PauseTime[6] := 0; END_IF;
   #DummyBool := NOT #CycleInStep[6] OR #CycleInStep[6];
END_REGION

REGION Network 27: Offset State
   // Boolean shows when a sequence is in Offset
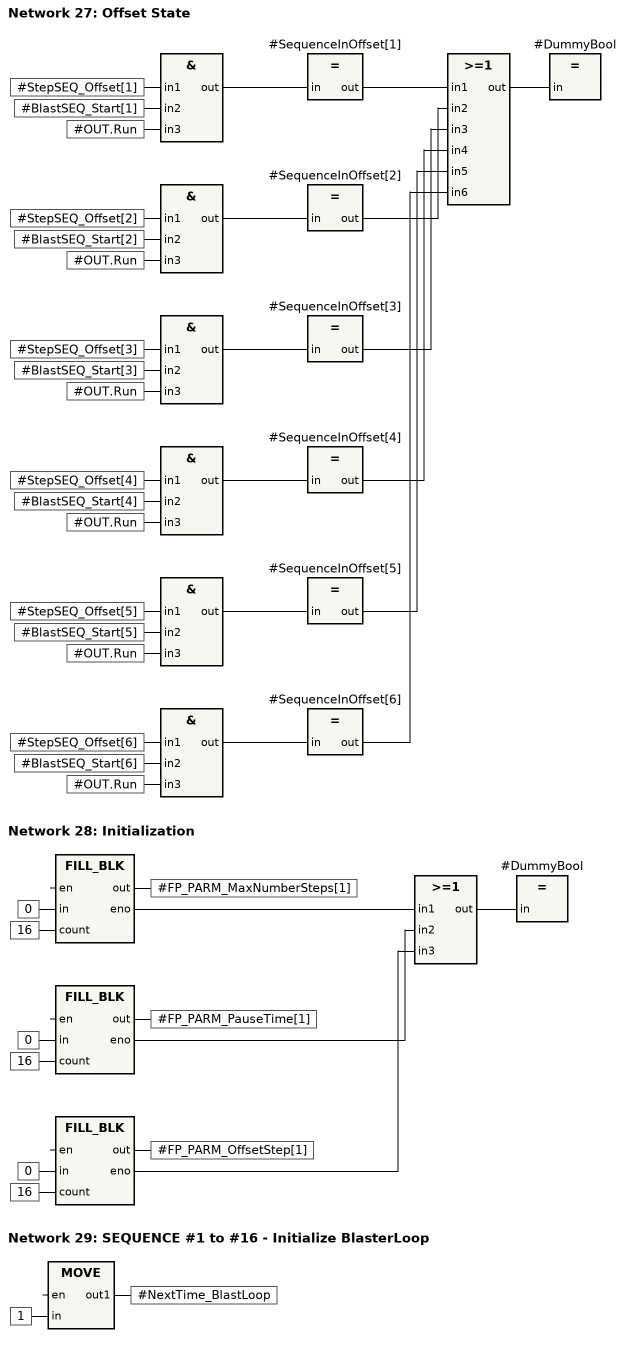
   #SequenceInOffset[1] := #StepSEQ_Offset[1] AND #BlastSEQ_Start[1] AND #OUT.Run;
   #SequenceInOffset[2] := #StepSEQ_Offset[2] AND #BlastSEQ_Start[2] AND #OUT.Run;
   #SequenceInOffset[3] := #StepSEQ_Offset[3] AND #BlastSEQ_Start[3] AND #OUT.Run;
   #SequenceInOffset[4] := #StepSEQ_Offset[4] AND #BlastSEQ_Start[4] AND #OUT.Run;
   #SequenceInOffset[5] := #StepSEQ_Offset[5] AND #BlastSEQ_Start[5] AND #OUT.Run;
   #SequenceInOffset[6] := #StepSEQ_Offset[6] AND #BlastSEQ_Start[6] AND #OUT.Run;
   #DummyBool := (#StepSEQ_Offset[1] AND #BlastSEQ_Start[1] AND #OUT.Run) OR (#StepSEQ_Offset[2] AND #BlastSEQ_Start[2] AND #OUT.Run) OR (#StepSEQ_Offset[3] AND #BlastSEQ_Start[3] AND #OUT.Run) OR (#StepSEQ_Offset[4] AND #BlastSEQ_Start[4] AND #OUT.Run) OR (#StepSEQ_Offset[5] AND #BlastSEQ_Start[5] AND #OUT.Run) OR (#StepSEQ_Offset[6] AND #BlastSEQ_Start[6] AND #OUT.Run);
END_REGION

REGION Network 28: Initialization
   FILL_BLK(IN := 0, COUNT := 16, OUT => #FP_PARM_MaxNumberSteps[1]);
   FILL_BLK(IN := 0, COUNT := 16, OUT => #FP_PARM_PauseTime[1]);
   FILL_BLK(IN := 0, COUNT := 16, OUT => #FP_PARM_OffsetStep[1]);
   #DummyBool := TRUE OR TRUE OR TRUE;
END_REGION

REGION Network 29: SEQUENCE #1 to #16 - Initialize BlasterLoop
   #NextTime_BlastLoop := 1;
END_REGION

REGION Network 30: Bs1: SEQUENCE #1 - Move Maximum Step Number, Pause Time and Offset State from Sequence to Blasters
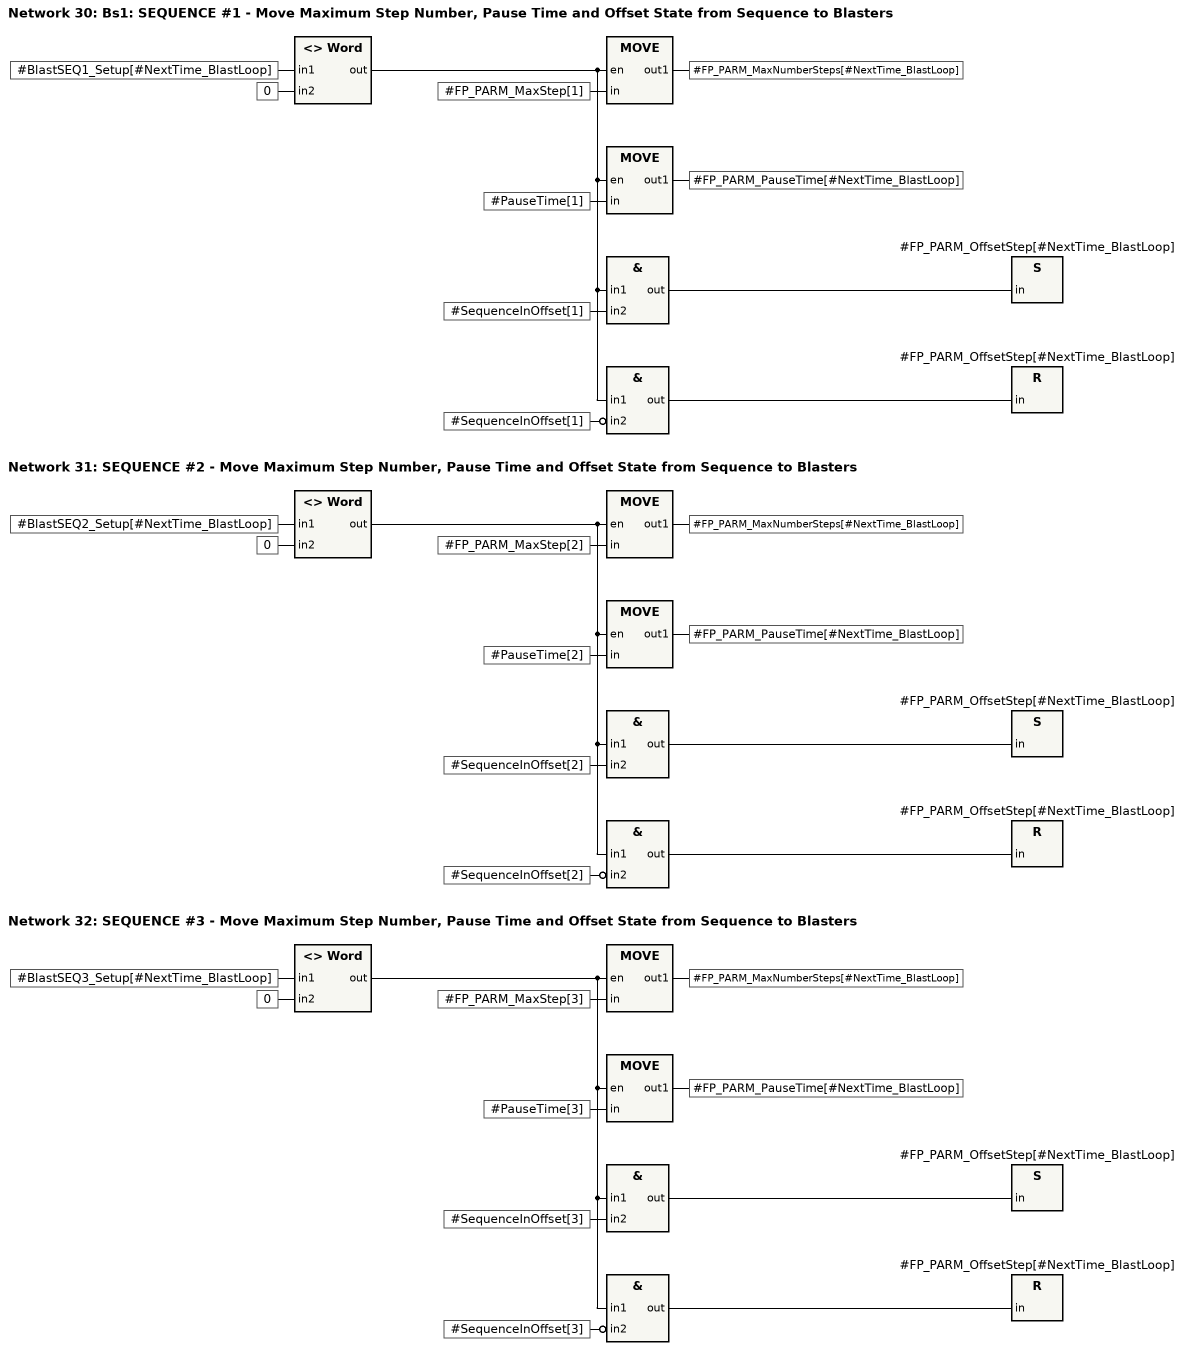
   Bs1:
   #_w1 := #BlastSEQ1_Setup[#NextTime_BlastLoop] <> 0;
   IF #_w1 THEN
       #FP_PARM_MaxNumberSteps[#NextTime_BlastLoop] := #FP_PARM_MaxStep[1];
       #FP_PARM_PauseTime[#NextTime_BlastLoop] := #PauseTime[1];
   END_IF;
   IF #_w1 AND #SequenceInOffset[1] THEN #FP_PARM_OffsetStep[#NextTime_BlastLoop] := TRUE; END_IF;
   IF #_w1 AND NOT #SequenceInOffset[1] THEN #FP_PARM_OffsetStep[#NextTime_BlastLoop] := FALSE; END_IF;
END_REGION

REGION Network 31: SEQUENCE #2 - Move Maximum Step Number, Pause Time and Offset State from Sequence to Blasters
   #_w1 := #BlastSEQ2_Setup[#NextTime_BlastLoop] <> 0;
   IF #_w1 THEN
       #FP_PARM_MaxNumberSteps[#NextTime_BlastLoop] := #FP_PARM_MaxStep[2];
       #FP_PARM_PauseTime[#NextTime_BlastLoop] := #PauseTime[2];
   END_IF;
   IF #_w1 AND #SequenceInOffset[2] THEN #FP_PARM_OffsetStep[#NextTime_BlastLoop] := TRUE; END_IF;
   IF #_w1 AND NOT #SequenceInOffset[2] THEN #FP_PARM_OffsetStep[#NextTime_BlastLoop] := FALSE; END_IF;
END_REGION

REGION Network 32: SEQUENCE #3 - Move Maximum Step Number, Pause Time and Offset State from Sequence to Blasters
   #_w1 := #BlastSEQ3_Setup[#NextTime_BlastLoop] <> 0;
   IF #_w1 THEN
       #FP_PARM_MaxNumberSteps[#NextTime_BlastLoop] := #FP_PARM_MaxStep[3];
       #FP_PARM_PauseTime[#NextTime_BlastLoop] := #PauseTime[3];
   END_IF;
   IF #_w1 AND #SequenceInOffset[3] THEN #FP_PARM_OffsetStep[#NextTime_BlastLoop] := TRUE; END_IF;
   IF #_w1 AND NOT #SequenceInOffset[3] THEN #FP_PARM_OffsetStep[#NextTime_BlastLoop] := FALSE; END_IF;
END_REGION

REGION Network 33: SEQUENCE #4 - Move Maximum Step Number, Pause Time and Offset State from Sequence to Blasters
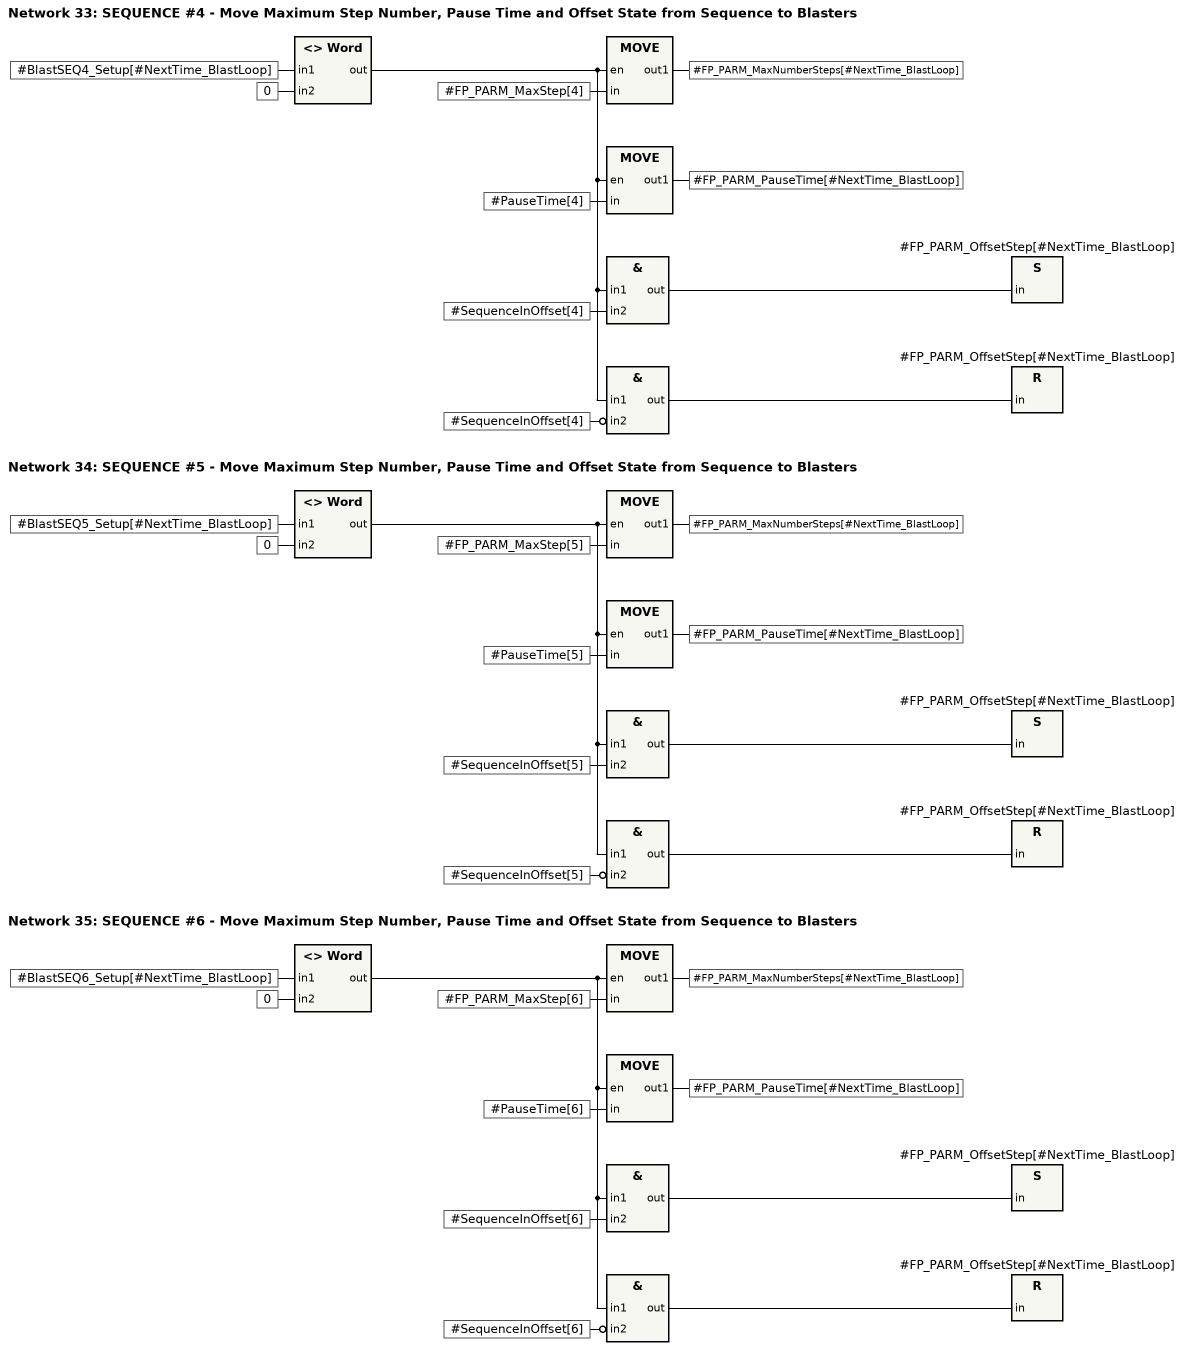
   #_w1 := #BlastSEQ4_Setup[#NextTime_BlastLoop] <> 0;
   IF #_w1 THEN
       #FP_PARM_MaxNumberSteps[#NextTime_BlastLoop] := #FP_PARM_MaxStep[4];
       #FP_PARM_PauseTime[#NextTime_BlastLoop] := #PauseTime[4];
   END_IF;
   IF #_w1 AND #SequenceInOffset[4] THEN #FP_PARM_OffsetStep[#NextTime_BlastLoop] := TRUE; END_IF;
   IF #_w1 AND NOT #SequenceInOffset[4] THEN #FP_PARM_OffsetStep[#NextTime_BlastLoop] := FALSE; END_IF;
END_REGION

REGION Network 34: SEQUENCE #5 - Move Maximum Step Number, Pause Time and Offset State from Sequence to Blasters
   #_w1 := #BlastSEQ5_Setup[#NextTime_BlastLoop] <> 0;
   IF #_w1 THEN
       #FP_PARM_MaxNumberSteps[#NextTime_BlastLoop] := #FP_PARM_MaxStep[5];
       #FP_PARM_PauseTime[#NextTime_BlastLoop] := #PauseTime[5];
   END_IF;
   IF #_w1 AND #SequenceInOffset[5] THEN #FP_PARM_OffsetStep[#NextTime_BlastLoop] := TRUE; END_IF;
   IF #_w1 AND NOT #SequenceInOffset[5] THEN #FP_PARM_OffsetStep[#NextTime_BlastLoop] := FALSE; END_IF;
END_REGION

REGION Network 35: SEQUENCE #6 - Move Maximum Step Number, Pause Time and Offset State from Sequence to Blasters
   #_w1 := #BlastSEQ6_Setup[#NextTime_BlastLoop] <> 0;
   IF #_w1 THEN
       #FP_PARM_MaxNumberSteps[#NextTime_BlastLoop] := #FP_PARM_MaxStep[6];
       #FP_PARM_PauseTime[#NextTime_BlastLoop] := #PauseTime[6];
   END_IF;
   IF #_w1 AND #SequenceInOffset[6] THEN #FP_PARM_OffsetStep[#NextTime_BlastLoop] := TRUE; END_IF;
   IF #_w1 AND NOT #SequenceInOffset[6] THEN #FP_PARM_OffsetStep[#NextTime_BlastLoop] := FALSE; END_IF;
END_REGION

REGION Network 36: SEQUENCE #1 to #16- Next Blaster
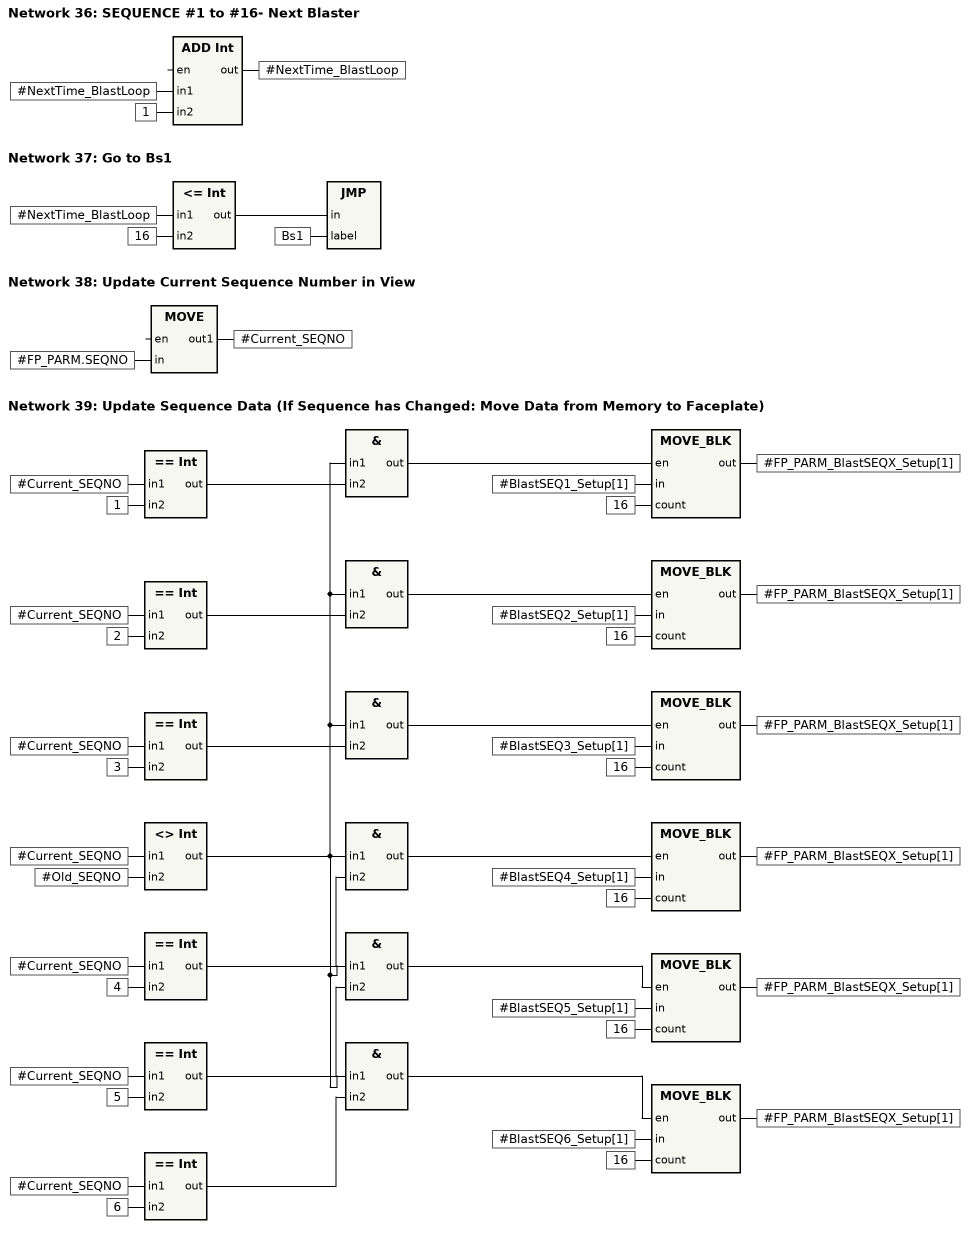
   #NextTime_BlastLoop := #NextTime_BlastLoop + 1;
END_REGION

REGION Network 37: Go to Bs1
   IF #NextTime_BlastLoop <= 16 THEN GOTO Bs1; END_IF;
END_REGION

REGION Network 38: Update Current Sequence Number in View
   #Current_SEQNO := #FP_PARM.SEQNO;
END_REGION

REGION Network 39: Update Sequence Data (If Sequence has Changed: Move Data from Memory to Faceplate)
   #_w1 := #Current_SEQNO <> #Old_SEQNO;
   IF #_w1 AND (#Current_SEQNO = 1) THEN
       MOVE_BLK(IN := #BlastSEQ1_Setup[1], COUNT := 16, OUT => #FP_PARM_BlastSEQX_Setup[1]);
   END_IF;
   IF #_w1 AND (#Current_SEQNO = 2) THEN
       MOVE_BLK(IN := #BlastSEQ2_Setup[1], COUNT := 16, OUT => #FP_PARM_BlastSEQX_Setup[1]);
   END_IF;
   IF #_w1 AND (#Current_SEQNO = 3) THEN
       MOVE_BLK(IN := #BlastSEQ3_Setup[1], COUNT := 16, OUT => #FP_PARM_BlastSEQX_Setup[1]);
   END_IF;
   IF #_w1 AND (#Current_SEQNO = 4) THEN
       MOVE_BLK(IN := #BlastSEQ4_Setup[1], COUNT := 16, OUT => #FP_PARM_BlastSEQX_Setup[1]);
   END_IF;
   IF #_w1 AND (#Current_SEQNO = 5) THEN
       MOVE_BLK(IN := #BlastSEQ5_Setup[1], COUNT := 16, OUT => #FP_PARM_BlastSEQX_Setup[1]);
   END_IF;
   IF #_w1 AND (#Current_SEQNO = 6) THEN
       MOVE_BLK(IN := #BlastSEQ6_Setup[1], COUNT := 16, OUT => #FP_PARM_BlastSEQX_Setup[1]);
   END_IF;
END_REGION

REGION Network 40: Update Sequence Data (Move Data from Faceplate to Memory)
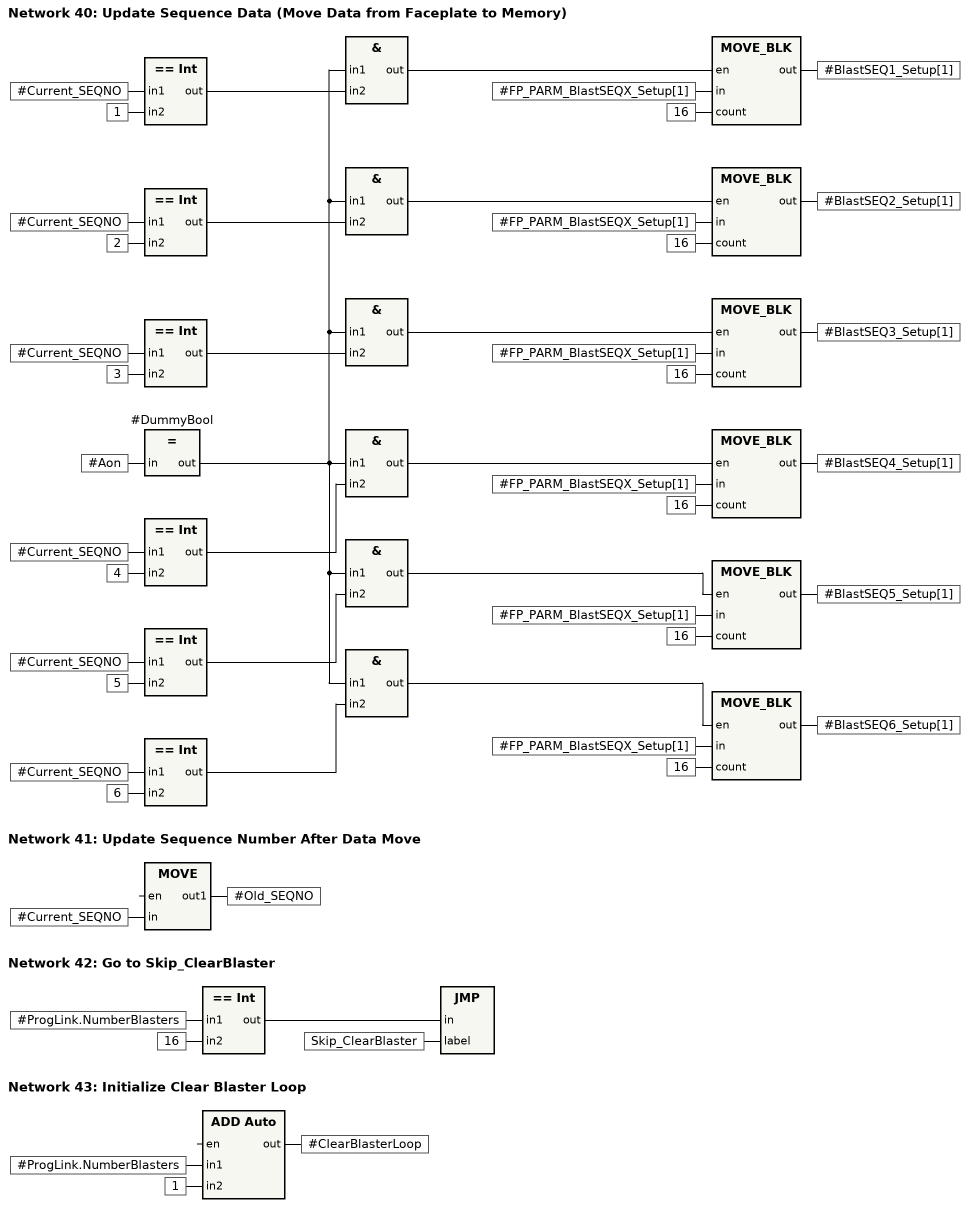
   #DummyBool := #Aon;
   IF #Aon AND (#Current_SEQNO = 1) THEN
       MOVE_BLK(IN := #FP_PARM_BlastSEQX_Setup[1], COUNT := 16, OUT => #BlastSEQ1_Setup[1]);
   END_IF;
   IF #Aon AND (#Current_SEQNO = 2) THEN
       MOVE_BLK(IN := #FP_PARM_BlastSEQX_Setup[1], COUNT := 16, OUT => #BlastSEQ2_Setup[1]);
   END_IF;
   IF #Aon AND (#Current_SEQNO = 3) THEN
       MOVE_BLK(IN := #FP_PARM_BlastSEQX_Setup[1], COUNT := 16, OUT => #BlastSEQ3_Setup[1]);
   END_IF;
   IF #Aon AND (#Current_SEQNO = 4) THEN
       MOVE_BLK(IN := #FP_PARM_BlastSEQX_Setup[1], COUNT := 16, OUT => #BlastSEQ4_Setup[1]);
   END_IF;
   IF #Aon AND (#Current_SEQNO = 5) THEN
       MOVE_BLK(IN := #FP_PARM_BlastSEQX_Setup[1], COUNT := 16, OUT => #BlastSEQ5_Setup[1]);
   END_IF;
   IF #Aon AND (#Current_SEQNO = 6) THEN
       MOVE_BLK(IN := #FP_PARM_BlastSEQX_Setup[1], COUNT := 16, OUT => #BlastSEQ6_Setup[1]);
   END_IF;
END_REGION

REGION Network 41: Update Sequence Number After Data Move
   // Update Memory Old_SEQNO with current SEQNO
   #Old_SEQNO := #Current_SEQNO;
END_REGION

REGION Network 42: Go to Skip_ClearBlaster
   IF #ProgLink.NumberBlasters = 16 THEN GOTO Skip_ClearBlaster; END_IF;
END_REGION

REGION Network 43: Initialize Clear Blaster Loop
   // Clearing starts with the blaster above the last configured
   #ClearBlasterLoop := #ProgLink.NumberBlasters + 1;
END_REGION

REGION Network 44: ClearBlaster
   // Clear configuration for unused Blasters in ECS Setup and in Stored Sequences 1-6
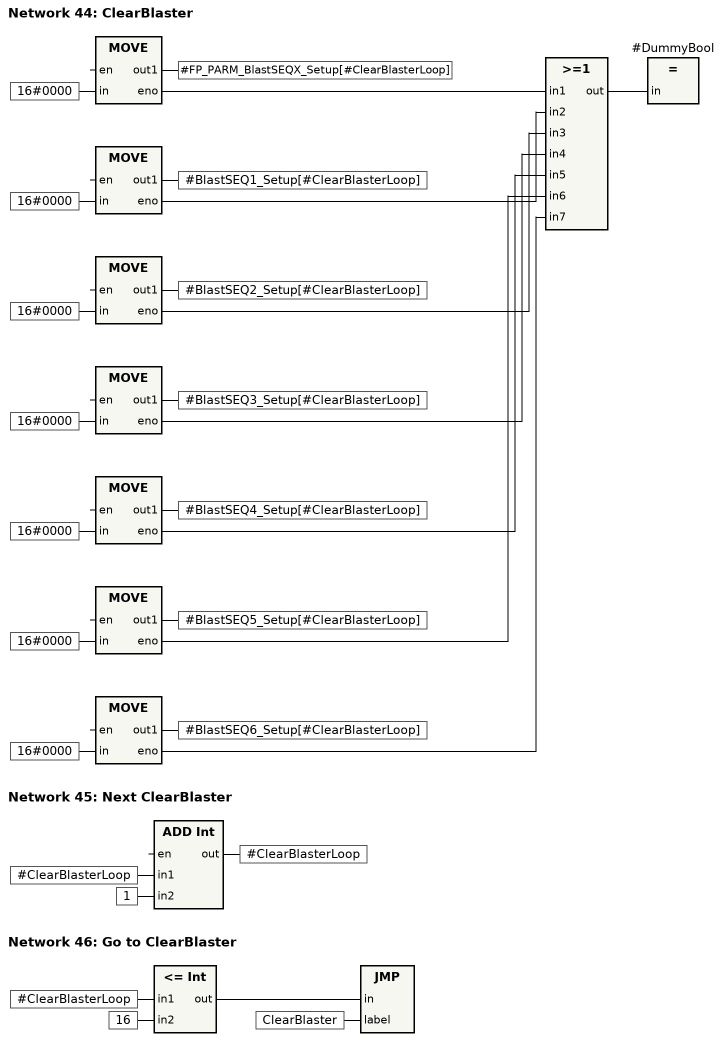
   ClearBlaster:
   #FP_PARM_BlastSEQX_Setup[#ClearBlasterLoop] := 16#0000;
   #BlastSEQ1_Setup[#ClearBlasterLoop] := 16#0000;
   #BlastSEQ2_Setup[#ClearBlasterLoop] := 16#0000;
   #BlastSEQ3_Setup[#ClearBlasterLoop] := 16#0000;
   #BlastSEQ4_Setup[#ClearBlasterLoop] := 16#0000;
   #BlastSEQ5_Setup[#ClearBlasterLoop] := 16#0000;
   #BlastSEQ6_Setup[#ClearBlasterLoop] := 16#0000;
   #DummyBool := TRUE OR TRUE OR TRUE OR TRUE OR TRUE OR TRUE OR TRUE;
END_REGION

REGION Network 45: Next ClearBlaster
   #ClearBlasterLoop := #ClearBlasterLoop + 1;
END_REGION

REGION Network 46: Go to ClearBlaster
   IF #ClearBlasterLoop <= 16 THEN GOTO ClearBlaster; END_IF;
END_REGION

REGION Network 47: Skip_ClearBlaster: Store Work Mask for Configured Number of Steps in the Program
   // StepMask: Allowed steps are set to 1
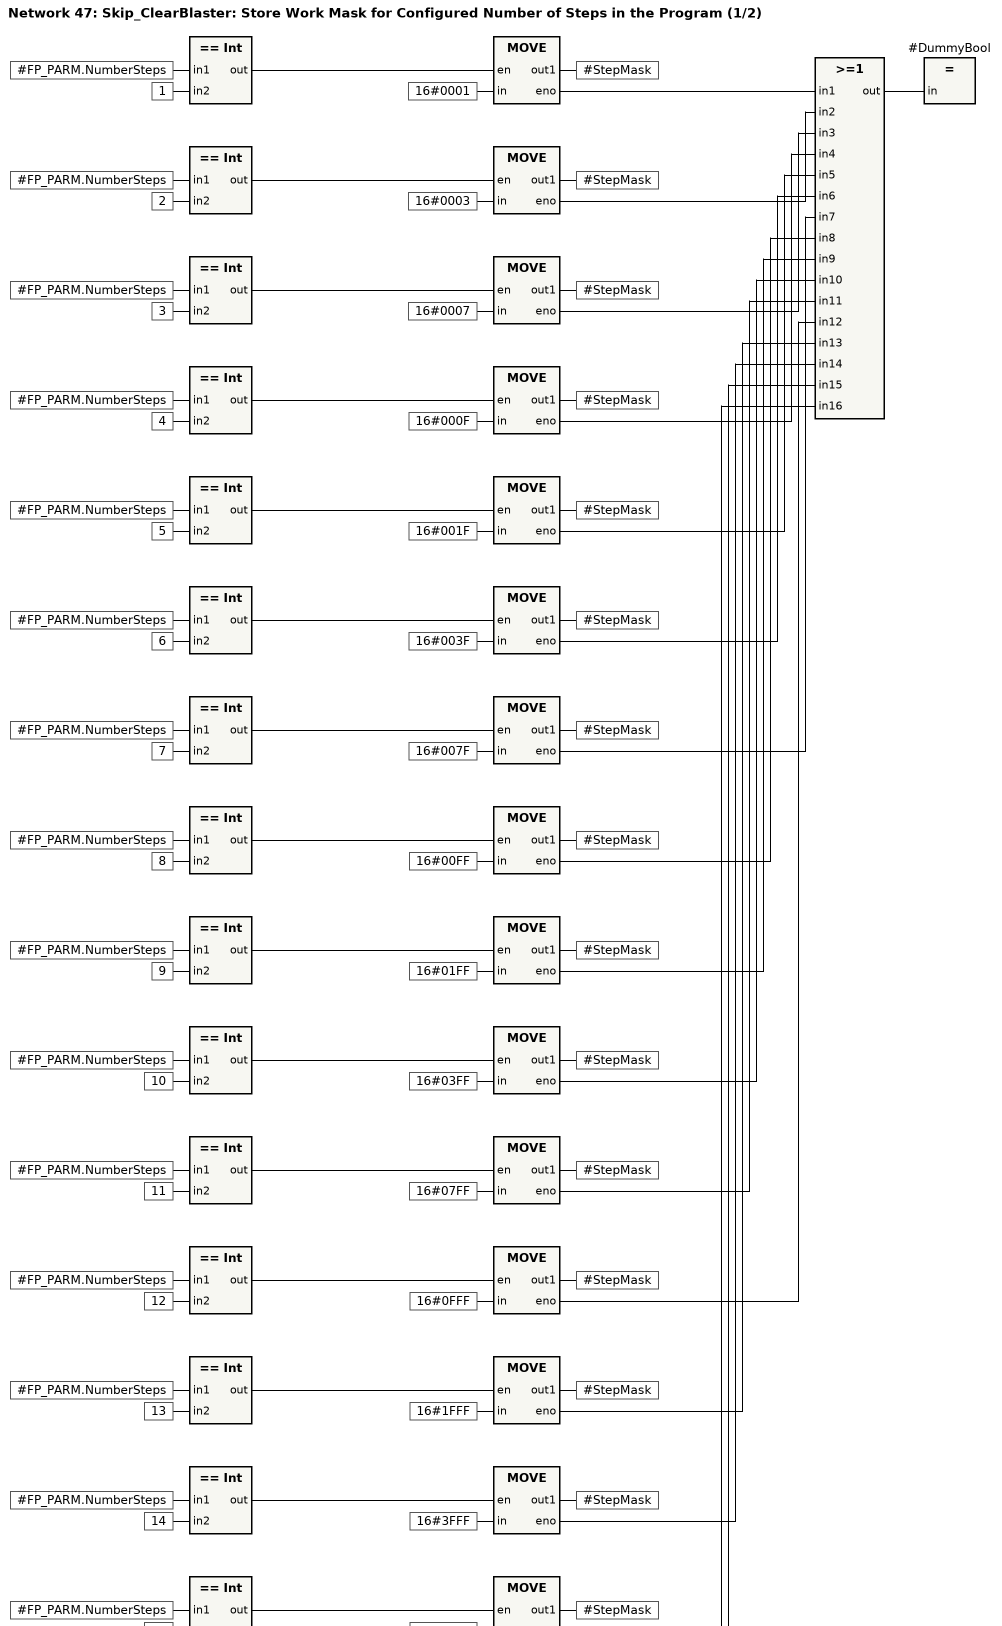
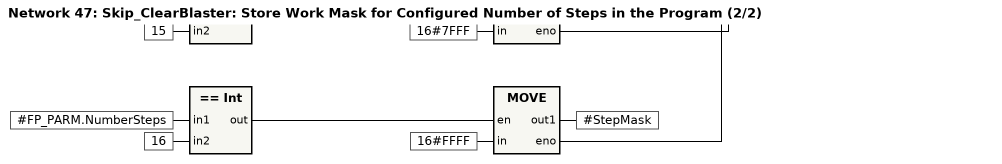
   Skip_ClearBlaster:
   #_w1 := #FP_PARM.NumberSteps = 1;
   IF #_w1 THEN #StepMask := 16#0001; END_IF;
   #_w2 := #FP_PARM.NumberSteps = 2;
   IF #_w2 THEN #StepMask := 16#0003; END_IF;
   #_w3 := #FP_PARM.NumberSteps = 3;
   IF #_w3 THEN #StepMask := 16#0007; END_IF;
   #_w4 := #FP_PARM.NumberSteps = 4;
   IF #_w4 THEN #StepMask := 16#000F; END_IF;
   #_w5 := #FP_PARM.NumberSteps = 5;
   IF #_w5 THEN #StepMask := 16#001F; END_IF;
   #_w6 := #FP_PARM.NumberSteps = 6;
   IF #_w6 THEN #StepMask := 16#003F; END_IF;
   #_w7 := #FP_PARM.NumberSteps = 7;
   IF #_w7 THEN #StepMask := 16#007F; END_IF;
   #_w8 := #FP_PARM.NumberSteps = 8;
   IF #_w8 THEN #StepMask := 16#00FF; END_IF;
   #_w9 := #FP_PARM.NumberSteps = 9;
   IF #_w9 THEN #StepMask := 16#01FF; END_IF;
   #_w10 := #FP_PARM.NumberSteps = 10;
   IF #_w10 THEN #StepMask := 16#03FF; END_IF;
   #_w11 := #FP_PARM.NumberSteps = 11;
   IF #_w11 THEN #StepMask := 16#07FF; END_IF;
   #_w12 := #FP_PARM.NumberSteps = 12;
   IF #_w12 THEN #StepMask := 16#0FFF; END_IF;
   #_w13 := #FP_PARM.NumberSteps = 13;
   IF #_w13 THEN #StepMask := 16#1FFF; END_IF;
   #_w14 := #FP_PARM.NumberSteps = 14;
   IF #_w14 THEN #StepMask := 16#3FFF; END_IF;
   #_w15 := #FP_PARM.NumberSteps = 15;
   IF #_w15 THEN #StepMask := 16#7FFF; END_IF;
   #_w16 := #FP_PARM.NumberSteps = 16;
   IF #_w16 THEN #StepMask := 16#FFFF; END_IF;
   #DummyBool := #_w1 OR #_w2 OR #_w3 OR #_w4 OR #_w5 OR #_w6 OR #_w7 OR #_w8 OR #_w9 OR #_w10 OR #_w11 OR #_w12 OR #_w13 OR #_w14 OR #_w15 OR #_w16;
END_REGION

REGION Network 48: Go to Skip_ClearSteps
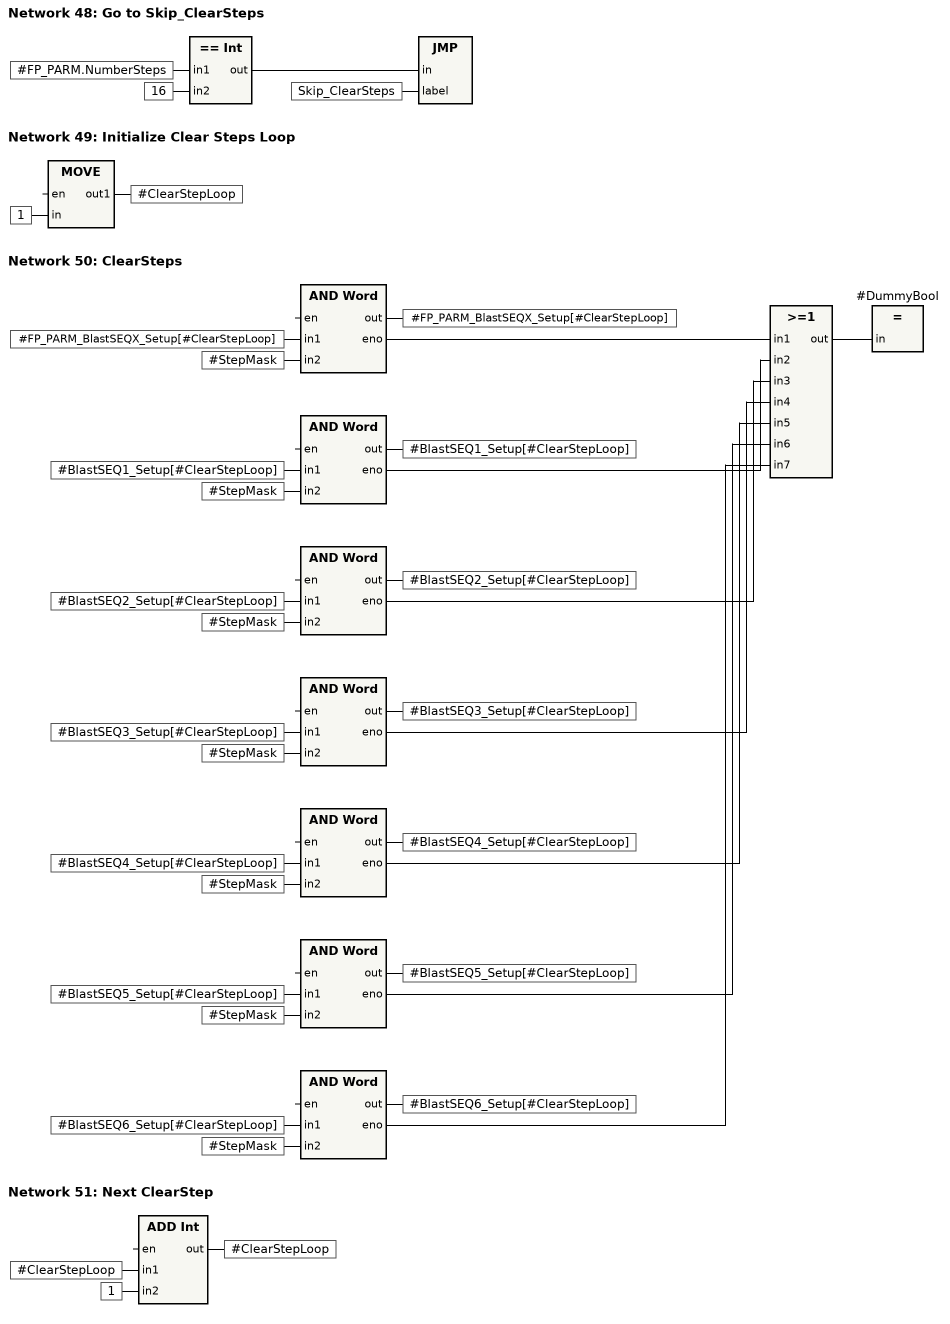
   IF #FP_PARM.NumberSteps = 16 THEN GOTO Skip_ClearSteps; END_IF;
END_REGION

REGION Network 49: Initialize Clear Steps Loop
   #ClearStepLoop := 1;
END_REGION

REGION Network 50: ClearSteps
   // Clear configuration for unused Steps in ECS Setup and in Stored Sequences 1-6
   ClearSteps:
   #FP_PARM_BlastSEQX_Setup[#ClearStepLoop] := #FP_PARM_BlastSEQX_Setup[#ClearStepLoop] AND #StepMask;
   #BlastSEQ1_Setup[#ClearStepLoop] := #BlastSEQ1_Setup[#ClearStepLoop] AND #StepMask;
   #BlastSEQ2_Setup[#ClearStepLoop] := #BlastSEQ2_Setup[#ClearStepLoop] AND #StepMask;
   #BlastSEQ3_Setup[#ClearStepLoop] := #BlastSEQ3_Setup[#ClearStepLoop] AND #StepMask;
   #BlastSEQ4_Setup[#ClearStepLoop] := #BlastSEQ4_Setup[#ClearStepLoop] AND #StepMask;
   #BlastSEQ5_Setup[#ClearStepLoop] := #BlastSEQ5_Setup[#ClearStepLoop] AND #StepMask;
   #BlastSEQ6_Setup[#ClearStepLoop] := #BlastSEQ6_Setup[#ClearStepLoop] AND #StepMask;
   #DummyBool := TRUE OR TRUE OR TRUE OR TRUE OR TRUE OR TRUE OR TRUE;
END_REGION

REGION Network 51: Next ClearStep
   #ClearStepLoop := #ClearStepLoop + 1;
END_REGION

REGION Network 52: Go to ClearSteps
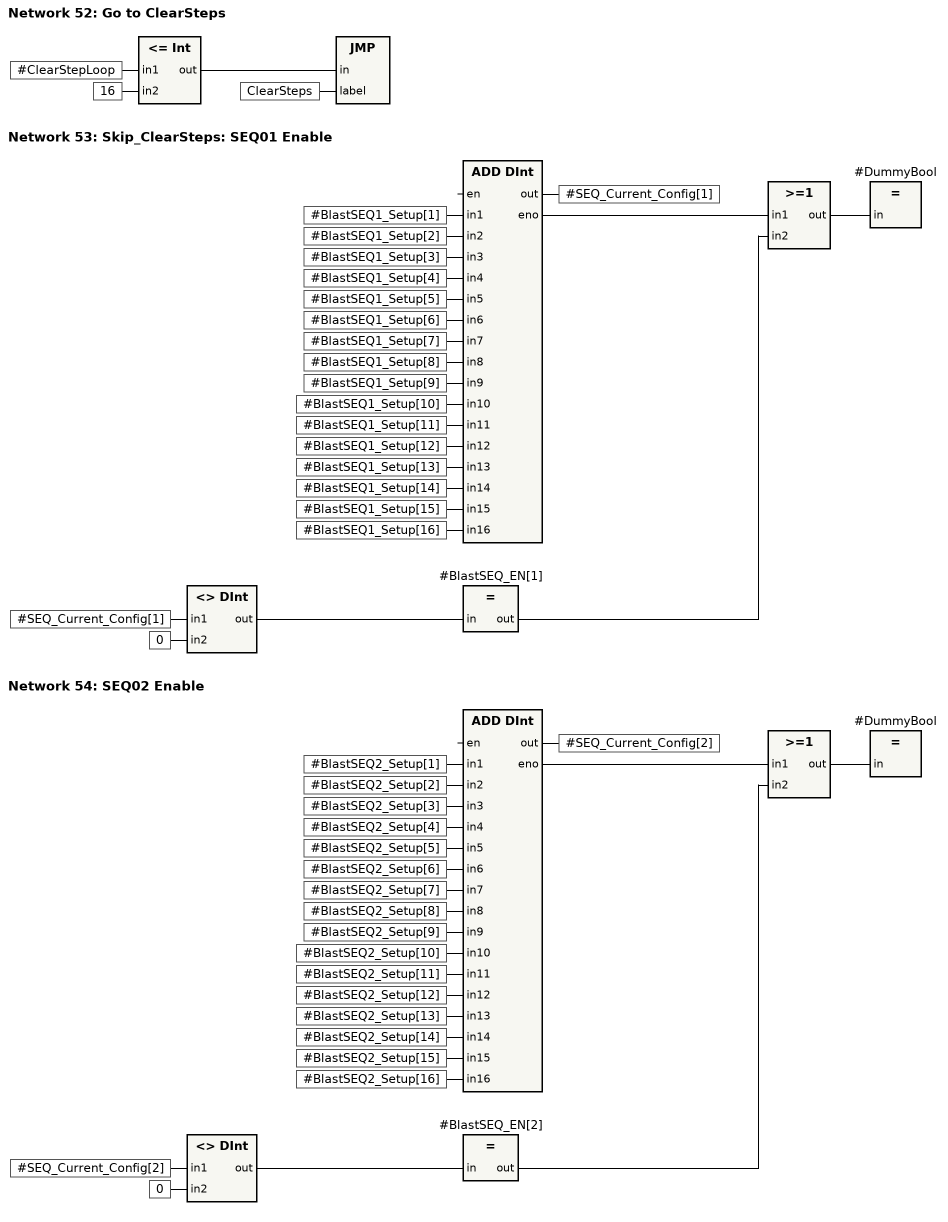
   IF #ClearStepLoop <= 16 THEN GOTO ClearSteps; END_IF;
END_REGION

REGION Network 53: Skip_ClearSteps: SEQ01 Enable
   Skip_ClearSteps:
   #SEQ_Current_Config[1] := #BlastSEQ1_Setup[1] + #BlastSEQ1_Setup[2] + #BlastSEQ1_Setup[3] + #BlastSEQ1_Setup[4] + #BlastSEQ1_Setup[5] + #BlastSEQ1_Setup[6] + #BlastSEQ1_Setup[7] + #BlastSEQ1_Setup[8] + #BlastSEQ1_Setup[9] + #BlastSEQ1_Setup[10] + #BlastSEQ1_Setup[11] + #BlastSEQ1_Setup[12] + #BlastSEQ1_Setup[13] + #BlastSEQ1_Setup[14] + #BlastSEQ1_Setup[15] + #BlastSEQ1_Setup[16];
   #BlastSEQ_EN[1] := #SEQ_Current_Config[1] <> 0;
   #DummyBool := TRUE OR (#SEQ_Current_Config[1] <> 0);
END_REGION

REGION Network 54: SEQ02 Enable
   #SEQ_Current_Config[2] := #BlastSEQ2_Setup[1] + #BlastSEQ2_Setup[2] + #BlastSEQ2_Setup[3] + #BlastSEQ2_Setup[4] + #BlastSEQ2_Setup[5] + #BlastSEQ2_Setup[6] + #BlastSEQ2_Setup[7] + #BlastSEQ2_Setup[8] + #BlastSEQ2_Setup[9] + #BlastSEQ2_Setup[10] + #BlastSEQ2_Setup[11] + #BlastSEQ2_Setup[12] + #BlastSEQ2_Setup[13] + #BlastSEQ2_Setup[14] + #BlastSEQ2_Setup[15] + #BlastSEQ2_Setup[16];
   #BlastSEQ_EN[2] := #SEQ_Current_Config[2] <> 0;
   #DummyBool := TRUE OR (#SEQ_Current_Config[2] <> 0);
END_REGION

REGION Network 55: SEQ03 Enable
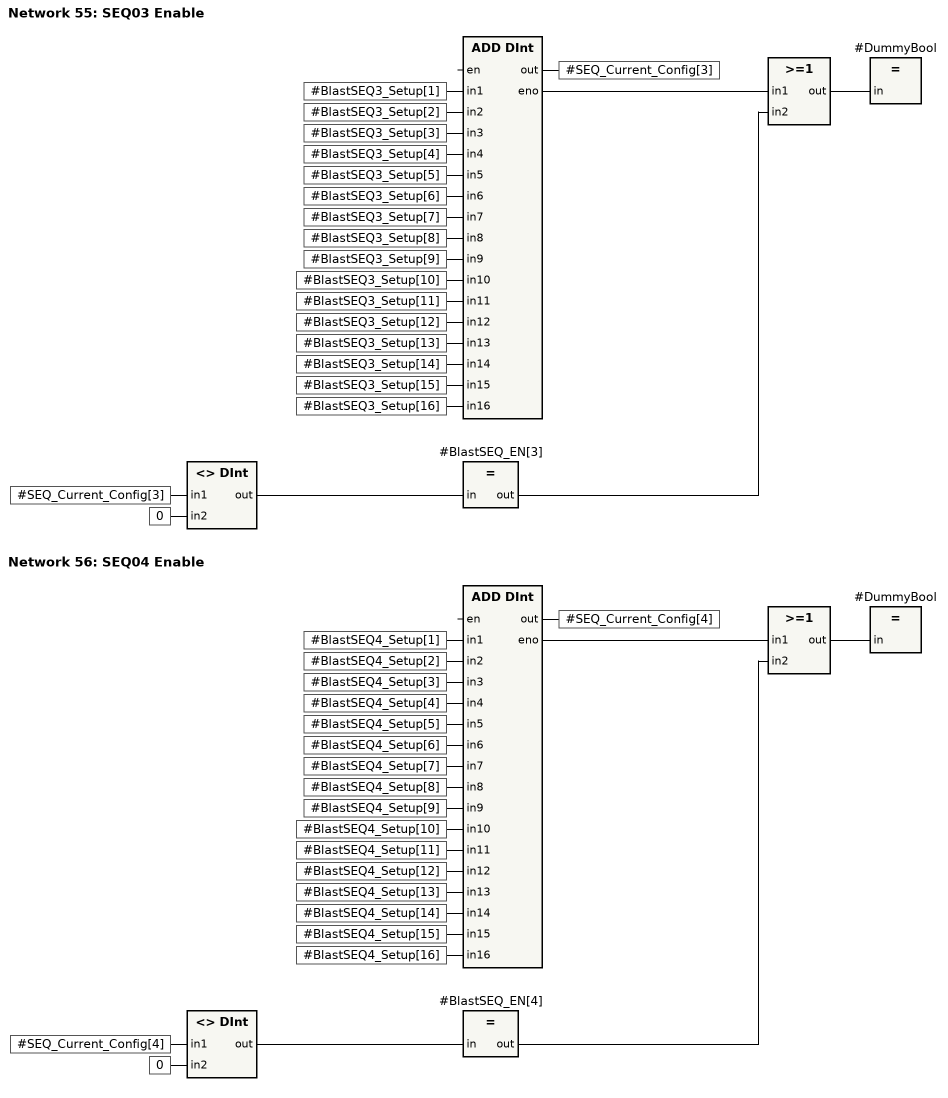
   #SEQ_Current_Config[3] := #BlastSEQ3_Setup[1] + #BlastSEQ3_Setup[2] + #BlastSEQ3_Setup[3] + #BlastSEQ3_Setup[4] + #BlastSEQ3_Setup[5] + #BlastSEQ3_Setup[6] + #BlastSEQ3_Setup[7] + #BlastSEQ3_Setup[8] + #BlastSEQ3_Setup[9] + #BlastSEQ3_Setup[10] + #BlastSEQ3_Setup[11] + #BlastSEQ3_Setup[12] + #BlastSEQ3_Setup[13] + #BlastSEQ3_Setup[14] + #BlastSEQ3_Setup[15] + #BlastSEQ3_Setup[16];
   #BlastSEQ_EN[3] := #SEQ_Current_Config[3] <> 0;
   #DummyBool := TRUE OR (#SEQ_Current_Config[3] <> 0);
END_REGION

REGION Network 56: SEQ04 Enable
   #SEQ_Current_Config[4] := #BlastSEQ4_Setup[1] + #BlastSEQ4_Setup[2] + #BlastSEQ4_Setup[3] + #BlastSEQ4_Setup[4] + #BlastSEQ4_Setup[5] + #BlastSEQ4_Setup[6] + #BlastSEQ4_Setup[7] + #BlastSEQ4_Setup[8] + #BlastSEQ4_Setup[9] + #BlastSEQ4_Setup[10] + #BlastSEQ4_Setup[11] + #BlastSEQ4_Setup[12] + #BlastSEQ4_Setup[13] + #BlastSEQ4_Setup[14] + #BlastSEQ4_Setup[15] + #BlastSEQ4_Setup[16];
   #BlastSEQ_EN[4] := #SEQ_Current_Config[4] <> 0;
   #DummyBool := TRUE OR (#SEQ_Current_Config[4] <> 0);
END_REGION

REGION Network 57: SEQ05 Enable
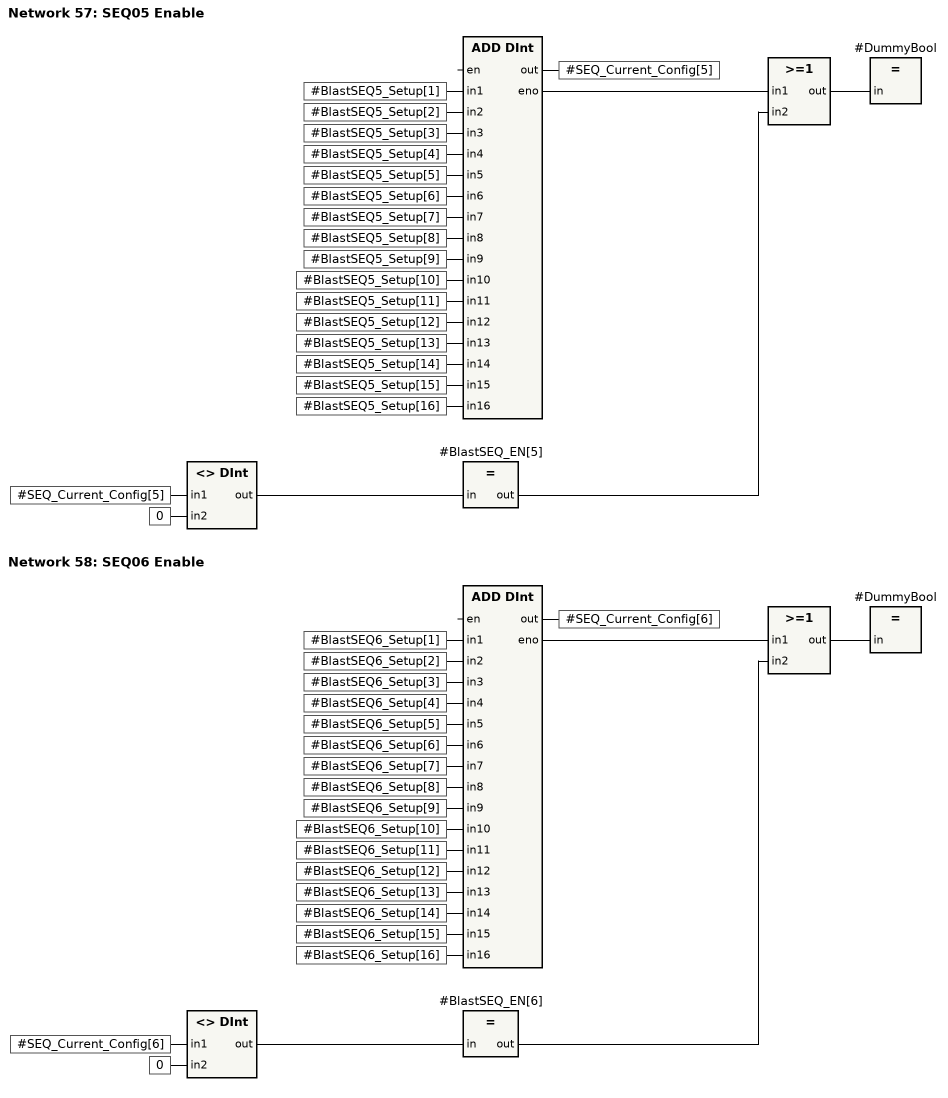
   #SEQ_Current_Config[5] := #BlastSEQ5_Setup[1] + #BlastSEQ5_Setup[2] + #BlastSEQ5_Setup[3] + #BlastSEQ5_Setup[4] + #BlastSEQ5_Setup[5] + #BlastSEQ5_Setup[6] + #BlastSEQ5_Setup[7] + #BlastSEQ5_Setup[8] + #BlastSEQ5_Setup[9] + #BlastSEQ5_Setup[10] + #BlastSEQ5_Setup[11] + #BlastSEQ5_Setup[12] + #BlastSEQ5_Setup[13] + #BlastSEQ5_Setup[14] + #BlastSEQ5_Setup[15] + #BlastSEQ5_Setup[16];
   #BlastSEQ_EN[5] := #SEQ_Current_Config[5] <> 0;
   #DummyBool := TRUE OR (#SEQ_Current_Config[5] <> 0);
END_REGION

REGION Network 58: SEQ06 Enable
   #SEQ_Current_Config[6] := #BlastSEQ6_Setup[1] + #BlastSEQ6_Setup[2] + #BlastSEQ6_Setup[3] + #BlastSEQ6_Setup[4] + #BlastSEQ6_Setup[5] + #BlastSEQ6_Setup[6] + #BlastSEQ6_Setup[7] + #BlastSEQ6_Setup[8] + #BlastSEQ6_Setup[9] + #BlastSEQ6_Setup[10] + #BlastSEQ6_Setup[11] + #BlastSEQ6_Setup[12] + #BlastSEQ6_Setup[13] + #BlastSEQ6_Setup[14] + #BlastSEQ6_Setup[15] + #BlastSEQ6_Setup[16];
   #BlastSEQ_EN[6] := #SEQ_Current_Config[6] <> 0;
   #DummyBool := TRUE OR (#SEQ_Current_Config[6] <> 0);
END_REGION

REGION Network 59: Go to NoChange_Setup
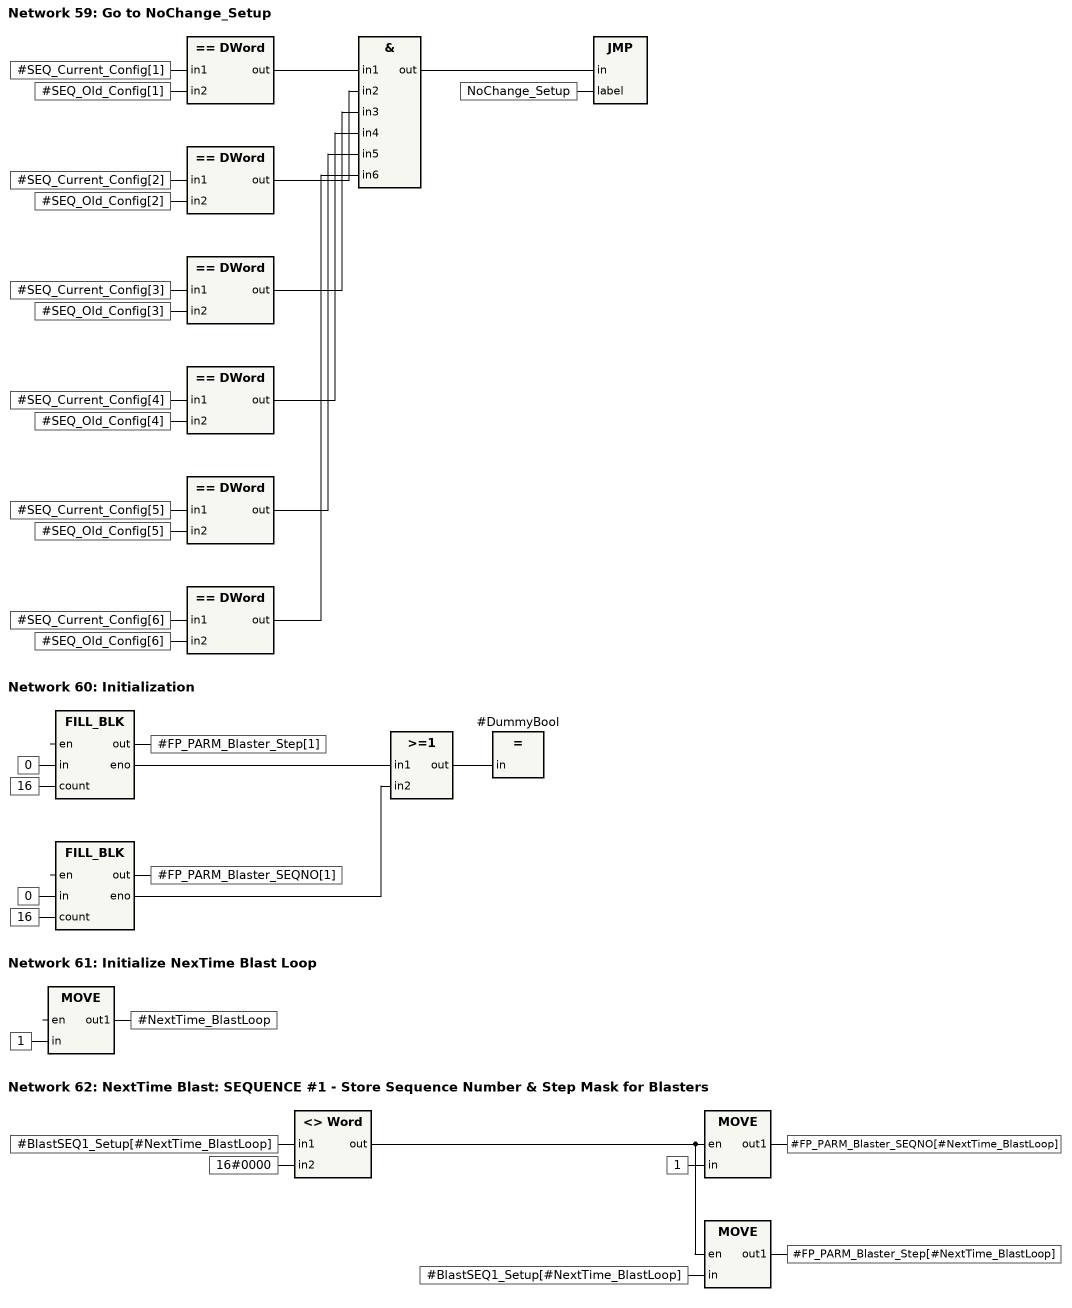
   IF (#SEQ_Current_Config[1] = #SEQ_Old_Config[1]) AND (#SEQ_Current_Config[2] = #SEQ_Old_Config[2]) AND (#SEQ_Current_Config[3] = #SEQ_Old_Config[3]) AND (#SEQ_Current_Config[4] = #SEQ_Old_Config[4]) AND (#SEQ_Current_Config[5] = #SEQ_Old_Config[5]) AND (#SEQ_Current_Config[6] = #SEQ_Old_Config[6]) THEN
       GOTO NoChange_Setup;
   END_IF;
END_REGION

REGION Network 60: Initialization
   FILL_BLK(IN := 0, COUNT := 16, OUT => #FP_PARM_Blaster_Step[1]);
   FILL_BLK(IN := 0, COUNT := 16, OUT => #FP_PARM_Blaster_SEQNO[1]);
   #DummyBool := TRUE OR TRUE;
END_REGION

REGION Network 61: Initialize NexTime Blast Loop
   #NextTime_BlastLoop := 1;
END_REGION

REGION Network 62: NextTime Blast: SEQUENCE #1 - Store Sequence Number & Step Mask for Blasters
   NexTimeBlast:
   #_w1 := #BlastSEQ1_Setup[#NextTime_BlastLoop] <> 16#0000;
   IF #_w1 THEN
       #FP_PARM_Blaster_SEQNO[#NextTime_BlastLoop] := 1;
       #FP_PARM_Blaster_Step[#NextTime_BlastLoop] := #BlastSEQ1_Setup[#NextTime_BlastLoop];
   END_IF;
END_REGION

REGION Network 63: SEQUENCE #2 - Store Sequence Number & Step Mask for Blasters
